C07286=1082.172,307.189,411.754,175.899,25.836,154.334
C07287=1082.167,306.941,411.785,175.896,25.832,154.333
C07288=1082.161,306.693,411.817,175.893,25.828,154.332
C07289=1082.155,306.445,411.848,175.890,25.824,154.332
C07290=1082.150,306.197,411.879,175.887,25.820,154.331
C07291=1082.144,305.949,411.911,175.885,25.816,154.331
C07292=1082.138,305.702,411.942,175.882,25.812,154.330
C07293=1082.132,305.453,411.973,175.879,25.808,154.330
C07294=1082.126,305.206,412.004,175.876,25.804,154.329
C07295=1082.121,304.958,412.036,175.873,25.800,154.328
C07296=1082.115,304.709,412.067,175.870,25.796,154.328
C07297=1082.109,304.462,412.098,175.867,25.792,154.327
C07298=1082.103,304.213,412.130,175.863,25.788,154.327
C07299=1082.093,303.800,412.182,175.859,25.781,154.326
C07300=1082.084,303.388,412.233,175.855,25.775,154.325
C07301=1082.075,302.974,412.286,175.849,25.768,154.324
C07302=1082.065,302.561,412.338,175.845,25.762,154.323
C07303=1082.059,302.314,412.368,175.842,25.758,154.323
C07304=1082.053,302.065,412.400,175.839,25.753,154.322
C07305=1082.047,301.818,412.430,175.836,25.749,154.321
C07306=1082.042,301.570,412.462,175.833,25.746,154.321
C07307=1082.037,301.322,412.493,175.831,25.742,154.320
C07308=1082.031,301.073,412.524,175.828,25.738,154.320
C07309=1082.025,300.826,412.555,175.825,25.734,154.319
C07310=1082.019,300.578,412.586,175.822,25.730,154.319
C07311=1082.014,300.330,412.617,175.818,25.726,154.318
C07312=1082.008,300.082,412.648,175.815,25.722,154.318
C07313=1082.002,299.834,412.679,175.813,25.718,154.317
C07314=1081.997,299.586,412.709,175.810,25.714,154.317
C07315=1081.991,299.339,412.741,175.807,25.710,154.316
C07316=1081.985,299.090,412.772,175.804,25.706,154.315
C07317=1081.980,298.842,412.803,175.801,25.702,154.315
C07318=1081.974,298.594,412.833,175.798,25.698,154.314
C07319=1081.969,298.346,412.864,175.796,25.695,154.314
C07320=1081.963,298.099,412.895,175.793,25.690,154.313
C07321=1081.957,297.850,412.926,175.790,25.686,154.313
C07322=1081.951,297.602,412.957,175.787,25.682,154.312
C07323=1081.945,297.354,412.987,175.784,25.678,154.312
C07324=1081.940,297.106,413.017,175.782,25.675,154.311
C07325=1081.934,296.858,413.049,175.779,25.671,154.310
C07326=1081.928,296.610,413.079,175.776,25.667,154.310
C07327=1081.922,296.362,413.109,175.773,25.663,154.309
C07328=1081.916,296.114,413.140,175.771,25.660,154.309
C07329=1081.910,295.866,413.172,175.767,25.656,154.308
C07330=1081.905,295.618,413.202,175.764,25.652,154.308
C07331=1081.899,295.370,413.232,175.761,25.648,154.307
C07332=1081.893,295.122,413.263,175.758,25.644,154.307
C07333=1081.887,294.875,413.293,175.756,25.641,154.306
C07334=1081.881,294.625,413.323,175.753,25.637,154.306
C07335=1081.875,294.378,413.353,175.750,25.633,154.305
C07336=1081.870,294.130,413.384,175.747,25.629,154.305
C07337=1081.864,293.882,413.415,175.744,25.625,154.304
C07338=1081.859,293.634,413.445,175.742,25.621,154.304
C07339=1081.853,293.386,413.475,175.739,25.618,154.303
C07340=1081.846,293.138,413.506,175.736,25.614,154.303
C07341=1081.841,292.890,413.537,175.733,25.610,154.302
C07342=1081.835,292.642,413.567,175.730,25.607,154.302
C07343=1081.829,292.393,413.597,175.727,25.603,154.301
C07344=1081.824,292.145,413.627,175.724,25.599,154.301
C07345=1081.818,291.897,413.658,175.721,25.595,154.300
C07346=1081.812,291.650,413.688,175.719,25.591,154.300
C07347=1081.806,291.401,413.719,175.716,25.588,154.299
C07348=1081.801,291.153,413.749,175.713,25.584,154.299
C07349=1081.795,290.905,413.779,175.710,25.580,154.298
C07350=1081.789,290.657,413.809,175.708,25.576,154.298
C07351=1081.780,290.258,413.858,175.703,25.570,154.297
C07352=1081.771,289.859,413.906,175.699,25.564,154.296
C07353=1081.761,289.460,413.955,175.694,25.558,154.295
C07354=1081.751,289.062,414.003,175.690,25.552,154.294
C07355=1081.746,288.813,414.032,175.687,25.548,154.294
C07356=1081.740,288.565,414.063,175.684,25.545,154.294
C07357=1081.734,288.318,414.093,175.681,25.541,154.293
C07358=1081.729,288.069,414.123,175.679,25.537,154.292
C07359=1081.723,287.821,414.153,175.675,25.533,154.292
C07360=1081.717,287.573,414.182,175.672,25.530,154.292
C07361=1081.711,287.325,414.212,175.670,25.526,154.291
C07362=1081.705,287.077,414.242,175.667,25.522,154.290
C07363=1081.699,286.829,414.272,175.664,25.519,154.290
C07364=1081.694,286.581,414.302,175.661,25.515,154.290
C07365=1081.688,286.333,414.332,175.659,25.511,154.289
C07366=1081.682,286.085,414.362,175.656,25.507,154.288
C07367=1081.676,285.837,414.392,175.653,25.504,154.288
C07368=1081.670,285.589,414.421,175.651,25.500,154.288
C07369=1081.665,285.340,414.451,175.648,25.496,154.287
C07370=1081.659,285.092,414.481,175.644,25.493,154.287
C07371=1081.653,284.844,414.511,175.641,25.489,154.286
C07372=1081.647,284.596,414.540,175.639,25.485,154.286
C07373=1081.642,284.348,414.571,175.636,25.482,154.285
C07374=1081.636,284.099,414.600,175.633,25.478,154.285
C07375=1081.631,283.851,414.630,175.631,25.474,154.284
C07376=1081.624,283.603,414.660,175.628,25.471,154.284
C07377=1081.618,283.355,414.689,175.625,25.467,154.283
C07378=1081.613,283.107,414.719,175.623,25.463,154.283
C07379=1081.607,282.859,414.749,175.620,25.460,154.282
C07380=1081.601,282.611,414.778,175.617,25.456,154.282
C07381=1081.595,282.362,414.808,175.614,25.452,154.281
C07382=1081.590,282.114,414.837,175.611,25.449,154.281
C07383=1081.584,281.865,414.867,175.608,25.445,154.280
C07384=1081.578,281.619,414.896,175.606,25.441,154.280
C07385=1081.573,281.370,414.926,175.603,25.438,154.279
C07386=1081.567,281.122,414.956,175.600,25.434,154.279
C07387=1081.561,280.873,414.985,175.598,25.430,154.278
C07388=1081.556,280.625,415.014,175.595,25.427,154.278
C07389=1081.550,280.377,415.044,175.592,25.423,154.277
C07390=1081.544,280.128,415.073,175.590,25.419,154.277
C07391=1081.538,279.881,415.103,175.587,25.416,154.276
C07392=1081.532,279.633,415.132,175.584,25.412,154.276
C07393=1081.526,279.384,415.162,175.581,25.408,154.275
C07394=1081.521,279.137,415.191,175.578,25.405,154.275
C07395=1081.515,278.888,415.220,175.575,25.401,154.274
C07396=1081.509,278.640,415.249,175.573,25.398,154.274
C07397=1081.503,278.392,415.279,175.570,25.394,154.274
C07398=1081.498,278.143,415.309,175.567,25.390,154.273
C07399=1081.492,277.895,415.338,175.565,25.387,154.273
C07400=1081.486,277.647,415.367,175.562,25.383,154.272
C07401=1081.481,277.399,415.395,175.559,25.379,154.272
C07402=1081.475,277.150,415.425,175.557,25.376,154.271
C07403=1081.466,276.762,415.471,175.552,25.370,154.270
C07404=1081.457,276.373,415.516,175.547,25.364,154.270
C07405=1081.448,275.983,415.562,175.544,25.359,154.269
C07406=1081.438,275.594,415.608,175.539,25.353,154.268
C07407=1081.434,275.346,415.637,175.536,25.349,154.268
C07408=1081.427,275.097,415.666,175.534,25.346,154.267
C07409=1081.421,274.849,415.695,175.531,25.342,154.267
C07410=1081.416,274.601,415.725,175.528,25.339,154.266
C07411=1081.410,274.353,415.753,175.526,25.335,154.266
C07412=1081.405,274.104,415.782,175.523,25.331,154.265
C07413=1081.399,273.856,415.811,175.520,25.328,154.265
C07414=1081.392,273.608,415.840,175.517,25.324,154.264
C07415=1081.388,273.360,415.869,175.514,25.321,154.264
C07416=1081.381,273.112,415.898,175.512,25.317,154.264
C07417=1081.375,272.863,415.927,175.509,25.314,154.263
C07418=1081.370,272.614,415.956,175.507,25.311,154.263
C07419=1081.364,272.367,415.984,175.504,25.307,154.262
C07420=1081.358,272.119,416.013,175.501,25.303,154.262
C07421=1081.352,271.870,416.042,175.499,25.300,154.261
C07422=1081.347,271.622,416.071,175.496,25.296,154.261
C07423=1081.341,271.374,416.100,175.493,25.292,154.260
C07424=1081.335,271.125,416.128,175.490,25.289,154.260
C07425=1081.329,270.877,416.157,175.487,25.285,154.259
C07426=1081.324,270.629,416.186,175.485,25.282,154.259
C07427=1081.318,270.381,416.215,175.482,25.278,154.259
C07428=1081.312,270.132,416.243,175.480,25.275,154.258
C07429=1081.306,269.885,416.272,175.477,25.271,154.258
C07430=1081.301,269.636,416.301,175.474,25.267,154.257
C07431=1081.295,269.387,416.330,175.472,25.264,154.257
C07432=1081.290,269.139,416.358,175.469,25.260,154.256
C07433=1081.283,268.891,416.387,175.466,25.257,154.256
C07434=1081.277,268.643,416.415,175.463,25.253,154.255
C07435=1081.272,268.394,416.443,175.460,25.250,154.255
C07436=1081.266,268.146,416.472,175.458,25.247,154.255
C07437=1081.261,267.897,416.501,175.455,25.243,154.254
C07438=1081.255,267.650,416.530,175.453,25.240,154.254
C07439=1081.249,267.401,416.558,175.450,25.236,154.253
C07440=1081.243,267.152,416.587,175.448,25.232,154.253
C07441=1081.237,266.905,416.615,175.445,25.229,154.252
C07442=1081.231,266.656,416.644,175.442,25.225,154.252
C07443=1081.226,266.408,416.672,175.439,25.222,154.251
C07444=1081.220,266.160,416.701,175.436,25.218,154.251
C07445=1081.214,265.911,416.729,175.434,25.215,154.250
C07446=1081.209,265.663,416.757,175.431,25.211,154.250
C07447=1081.203,265.414,416.785,175.429,25.208,154.250
C07448=1081.198,265.167,416.814,175.426,25.204,154.249
C07449=1081.192,264.918,416.843,175.424,25.201,154.249
C07450=1081.186,264.670,416.871,175.421,25.197,154.248
C07451=1081.180,264.421,416.899,175.418,25.193,154.248
C07452=1081.175,264.173,416.927,175.415,25.190,154.247
C07453=1081.169,263.924,416.955,175.412,25.186,154.247
C07454=1081.162,263.677,416.984,175.410,25.183,154.246
C07455=1081.154,263.290,417.027,175.406,25.178,154.246
C07456=1081.145,262.904,417.071,175.402,25.172,154.245
C07457=1081.135,262.518,417.115,175.397,25.167,154.244
C07458=1081.126,262.132,417.159,175.394,25.162,154.244
C07459=1081.120,261.883,417.187,175.390,25.158,154.243
C07460=1081.115,261.635,417.215,175.388,25.155,154.243
C07461=1081.108,261.387,417.243,175.385,25.151,154.242
C07462=1081.103,261.139,417.271,175.383,25.148,154.242
C07463=1081.097,260.890,417.299,175.380,25.144,154.242
C07464=1081.092,260.642,417.327,175.378,25.141,154.241
C07465=1081.085,260.393,417.355,175.375,25.137,154.241
C07466=1081.079,260.145,417.383,175.372,25.134,154.240
C07467=1081.074,259.897,417.411,175.370,25.131,154.240
C07468=1081.068,259.649,417.439,175.366,25.127,154.240
C07469=1081.062,259.400,417.467,175.364,25.124,154.239
C07470=1081.056,259.152,417.494,175.361,25.120,154.239
C07471=1081.051,258.903,417.522,175.359,25.117,154.238
C07472=1081.045,258.655,417.550,175.356,25.113,154.238
C07473=1081.039,258.406,417.578,175.354,25.110,154.237
C07474=1081.033,258.158,417.606,175.351,25.106,154.237
C07475=1081.027,257.909,417.634,175.349,25.103,154.236
C07476=1081.021,257.662,417.661,175.346,25.099,154.236
C07477=1081.016,257.412,417.689,175.343,25.096,154.236
C07478=1081.010,257.164,417.717,175.340,25.093,154.235
C07479=1081.004,256.916,417.745,175.338,25.089,154.235
C07480=1080.998,256.668,417.773,175.335,25.085,154.234
C07481=1080.993,256.419,417.800,175.333,25.082,154.234
C07482=1080.986,256.171,417.828,175.330,25.079,154.233
C07483=1080.981,255.923,417.856,175.328,25.075,154.233
C07484=1080.975,255.674,417.884,175.325,25.072,154.233
C07485=1080.969,255.426,417.911,175.322,25.068,154.232
C07486=1080.964,255.178,417.939,175.319,25.065,154.232
C07487=1080.958,254.929,417.967,175.317,25.061,154.231
C07488=1080.952,254.680,417.994,175.314,25.058,154.231
C07489=1080.946,254.432,418.022,175.312,25.055,154.230
C07490=1080.941,254.183,418.049,175.309,25.051,154.230
C07491=1080.935,253.935,418.077,175.307,25.048,154.229
C07492=1080.929,253.686,418.105,175.304,25.044,154.229
C07493=1080.924,253.438,418.132,175.302,25.041,154.229
C07494=1080.918,253.190,418.159,175.299,25.037,154.228
C07495=1080.913,252.941,418.187,175.296,25.034,154.228
C07496=1080.906,252.693,418.214,175.294,25.031,154.227
C07497=1080.901,252.444,418.242,175.291,25.027,154.227
C07498=1080.896,252.196,418.270,175.289,25.023,154.226
C07499=1080.890,251.947,418.297,175.286,25.020,154.226
C07500=1080.884,251.699,418.325,175.284,25.016,154.226
C07501=1080.879,251.451,418.351,175.281,25.013,154.225
C07502=1080.873,251.202,418.380,175.279,25.010,154.225
C07503=1080.868,250.953,418.407,175.276,25.006,154.224
C07504=1080.862,250.706,418.434,175.273,25.003,154.224
C07505=1080.857,250.457,418.461,175.270,24.999,154.223
C07506=1080.850,250.208,418.489,175.268,24.995,154.223
C07507=1080.842,249.820,418.532,175.265,24.990,154.222
C07508=1080.833,249.431,418.574,175.260,24.985,154.222
C07509=1080.824,249.042,418.617,175.256,24.979,154.221
C07510=1080.815,248.654,418.660,175.252,24.974,154.220
C07511=1080.810,248.404,418.687,175.250,24.970,154.220
C07512=1080.804,248.156,418.714,175.247,24.966,154.219
C07513=1080.799,247.908,418.742,175.245,24.963,154.219
C07514=1080.793,247.659,418.769,175.242,24.960,154.218
C07515=1080.788,247.411,418.796,175.239,24.956,154.218
C07516=1080.782,247.162,418.823,175.237,24.953,154.217
C07517=1080.776,246.914,418.851,175.234,24.949,154.217
C07518=1080.770,246.665,418.878,175.232,24.946,154.217
C07519=1080.765,246.417,418.904,175.229,24.942,154.216
C07520=1080.759,246.168,418.931,175.227,24.939,154.216
C07521=1080.754,245.920,418.958,175.225,24.936,154.215
C07522=1080.747,245.671,418.985,175.222,24.932,154.215
C07523=1080.742,245.423,419.013,175.220,24.929,154.214
C07524=1080.736,245.174,419.040,175.217,24.925,154.214
C07525=1080.730,244.926,419.066,175.214,24.922,154.214
C07526=1080.725,244.677,419.094,175.211,24.918,154.213
C07527=1080.720,244.429,419.120,175.209,24.915,154.213
C07528=1080.713,244.180,419.147,175.207,24.912,154.212
C07529=1080.707,243.932,419.174,175.204,24.908,154.212
C07530=1080.702,243.683,419.201,175.202,24.905,154.211
C07531=1080.697,243.435,419.228,175.199,24.901,154.211
C07532=1080.691,243.186,419.254,175.197,24.898,154.211
C07533=1080.686,242.937,419.282,175.194,24.895,154.210
C07534=1080.680,242.689,419.308,175.192,24.891,154.210
C07535=1080.674,242.441,419.335,175.189,24.888,154.209
C07536=1080.668,242.192,419.362,175.186,24.884,154.209
C07537=1080.662,241.943,419.389,175.184,24.881,154.209
C07538=1080.656,241.695,419.415,175.182,24.878,154.208
C07539=1080.651,241.447,419.442,175.179,24.874,154.208
C07540=1080.645,241.198,419.469,175.177,24.871,154.207
C07541=1080.640,240.950,419.496,175.174,24.867,154.207
C07542=1080.634,240.701,419.522,175.172,24.864,154.206
C07543=1080.628,240.453,419.549,175.169,24.861,154.206
C07544=1080.622,240.204,419.576,175.166,24.857,154.206
C07545=1080.616,239.955,419.602,175.164,24.853,154.205
C07546=1080.611,239.706,419.629,175.161,24.850,154.205
C07547=1080.605,239.458,419.655,175.159,24.847,154.204
C07548=1080.599,239.210,419.682,175.157,24.844,154.204
C07549=1080.593,238.961,419.709,175.154,24.840,154.204
C07550=1080.588,238.712,419.735,175.152,24.836,154.203
C07551=1080.582,238.464,419.761,175.150,24.833,154.203
C07552=1080.576,238.216,419.788,175.146,24.830,154.202
C07553=1080.571,237.967,419.815,175.144,24.827,154.202
C07554=1080.565,237.719,419.841,175.141,24.823,154.201
C07555=1080.559,237.470,419.867,175.139,24.820,154.201
C07556=1080.554,237.222,419.894,175.137,24.816,154.200
C07557=1080.548,236.973,419.920,175.134,24.813,154.200
C07558=1080.542,236.724,419.946,175.132,24.810,154.200
C07559=1080.533,236.329,419.989,175.128,24.804,154.199
C07560=1080.524,235.934,420.031,175.124,24.799,154.198
C07561=1080.515,235.538,420.073,175.120,24.793,154.198
C07562=1080.506,235.142,420.115,175.116,24.788,154.197
C07563=1080.500,234.893,420.141,175.113,24.784,154.197
C07564=1080.495,234.645,420.168,175.111,24.781,154.196
C07565=1080.489,234.396,420.194,175.108,24.777,154.196
C07566=1080.483,234.147,420.220,175.106,24.774,154.195
C07567=1080.478,233.899,420.246,175.104,24.771,154.195
C07568=1080.472,233.651,420.272,175.101,24.767,154.194
C07569=1080.466,233.402,420.298,175.099,24.764,154.194
C07570=1080.461,233.154,420.324,175.097,24.760,154.194
C07571=1080.455,232.905,420.350,175.094,24.757,154.193
C07572=1080.449,232.656,420.377,175.092,24.754,154.193
C07573=1080.444,232.407,420.403,175.089,24.751,154.192
C07574=1080.438,232.159,420.430,175.086,24.747,154.192
C07575=1080.432,231.910,420.455,175.084,24.743,154.191
C07576=1080.426,231.662,420.482,175.082,24.740,154.191
C07577=1080.421,231.413,420.508,175.079,24.737,154.191
C07578=1080.415,231.164,420.533,175.077,24.734,154.190
C07579=1080.410,230.916,420.560,175.075,24.730,154.190
C07580=1080.404,230.668,420.585,175.072,24.726,154.189
C07581=1080.398,230.419,420.612,175.070,24.723,154.189
C07582=1080.393,230.170,420.638,175.067,24.720,154.188
C07583=1080.387,229.921,420.664,175.064,24.716,154.188
C07584=1080.381,229.673,420.690,175.062,24.713,154.188
C07585=1080.375,229.424,420.716,175.060,24.710,154.187
C07586=1080.369,229.176,420.741,175.057,24.706,154.187
C07587=1080.364,228.927,420.767,175.055,24.703,154.186
C07588=1080.358,228.678,420.793,175.053,24.700,154.186
C07589=1080.352,228.430,420.818,175.051,24.696,154.186
C07590=1080.347,228.181,420.844,175.048,24.693,154.185
C07591=1080.341,227.932,420.870,175.045,24.690,154.185
C07592=1080.335,227.684,420.896,175.043,24.687,154.184
C07593=1080.329,227.435,420.922,175.040,24.683,154.184
C07594=1080.323,227.187,420.948,175.038,24.679,154.183
C07595=1080.318,226.938,420.973,175.036,24.676,154.183
C07596=1080.313,226.689,420.999,175.033,24.673,154.183
C07597=1080.307,226.441,421.024,175.031,24.669,154.182
C07598=1080.301,226.192,421.051,175.029,24.666,154.182
C07599=1080.295,225.944,421.076,175.027,24.663,154.181
C07600=1080.289,225.695,421.102,175.024,24.659,154.181
C07601=1080.283,225.447,421.127,175.022,24.656,154.181
C07602=1080.278,225.198,421.153,175.019,24.653,154.180
C07603=1080.273,224.949,421.179,175.016,24.649,154.180
C07604=1080.266,224.700,421.205,175.014,24.645,154.179
C07605=1080.261,224.452,421.230,175.012,24.642,154.179
C07606=1080.255,224.203,421.255,175.010,24.639,154.178
C07607=1080.250,223.954,421.281,175.007,24.636,154.178
C07608=1080.244,223.705,421.307,175.005,24.632,154.178
C07609=1080.239,223.457,421.332,175.003,24.629,154.177
C07610=1080.232,223.208,421.358,175.000,24.625,154.177
C07611=1080.224,222.805,421.399,174.996,24.620,154.176
C07612=1080.214,222.400,421.441,174.993,24.614,154.175
C07613=1080.205,221.996,421.483,174.988,24.609,154.175
C07614=1080.196,221.592,421.524,174.985,24.603,154.174
C07615=1080.190,221.343,421.550,174.982,24.600,154.174
C07616=1080.184,221.095,421.575,174.980,24.597,154.173
C07617=1080.179,220.847,421.600,174.977,24.593,154.173
C07618=1080.173,220.597,421.625,174.975,24.590,154.172
C07619=1080.167,220.349,421.651,174.973,24.587,154.172
C07620=1080.161,220.100,421.676,174.971,24.583,154.172
C07621=1080.155,219.852,421.701,174.968,24.580,154.171
C07622=1080.150,219.603,421.727,174.966,24.577,154.171
C07623=1080.144,219.354,421.752,174.964,24.573,154.170
C07624=1080.139,219.106,421.776,174.962,24.570,154.170
C07625=1080.133,218.857,421.802,174.959,24.566,154.169
C07626=1080.127,218.608,421.828,174.956,24.563,154.169
C07627=1080.121,218.360,421.853,174.954,24.560,154.169
C07628=1080.116,218.110,421.878,174.952,24.557,154.168
C07629=1080.110,217.862,421.903,174.949,24.553,154.168
C07630=1080.104,217.614,421.928,174.947,24.549,154.167
C07631=1080.098,217.365,421.953,174.945,24.546,154.167
C07632=1080.093,217.116,421.979,174.943,24.543,154.166
C07633=1080.087,216.868,422.004,174.940,24.539,154.166
C07634=1080.081,216.618,422.028,174.938,24.536,154.166
C07635=1080.076,216.370,422.053,174.936,24.533,154.165
C07636=1080.070,216.121,422.079,174.934,24.529,154.165
C07637=1080.064,215.872,422.104,174.930,24.526,154.164
C07638=1080.059,215.624,422.129,174.928,24.523,154.164
C07639=1080.053,215.375,422.154,174.926,24.519,154.164
C07640=1080.048,215.127,422.179,174.924,24.516,154.163
C07641=1080.042,214.878,422.204,174.921,24.512,154.163
C07642=1080.037,214.629,422.229,174.919,24.509,154.162
C07643=1080.030,214.381,422.254,174.917,24.506,154.162
C07644=1080.024,214.131,422.279,174.915,24.503,154.161
C07645=1080.020,213.883,422.304,174.913,24.499,154.161
C07646=1080.013,213.634,422.329,174.910,24.495,154.161
C07647=1080.008,213.386,422.354,174.908,24.492,154.160
C07648=1080.002,213.137,422.379,174.905,24.489,154.160
C07649=1079.997,212.889,422.403,174.903,24.486,154.159
C07650=1079.991,212.639,422.428,174.900,24.482,154.159
C07651=1079.986,212.391,422.453,174.898,24.478,154.158
C07652=1079.980,212.142,422.478,174.896,24.475,154.158
C07653=1079.974,211.894,422.503,174.894,24.472,154.158
C07654=1079.968,211.644,422.528,174.892,24.469,154.157
C07655=1079.963,211.396,422.553,174.889,24.465,154.157
C07656=1079.957,211.147,422.577,174.887,24.461,154.156
C07657=1079.952,210.899,422.602,174.885,24.458,154.156
C07658=1079.945,210.650,422.627,174.883,24.455,154.156
C07659=1079.940,210.401,422.651,174.881,24.452,154.155
C07660=1079.934,210.152,422.676,174.877,24.448,154.155
C07661=1079.929,209.904,422.701,174.875,24.445,154.154
C07662=1079.923,209.655,422.725,174.873,24.441,154.154
C07663=1079.913,209.254,422.765,174.870,24.436,154.153
C07664=1079.905,208.855,422.804,174.866,24.431,154.153
C07665=1079.895,208.455,422.844,174.863,24.425,154.152
C07666=1079.886,208.055,422.884,174.859,24.420,154.151
C07667=1079.863,207.021,422.983,174.758,24.366,154.153
C07668=1079.856,206.772,423.007,174.755,24.364,154.153
C07669=1079.851,206.523,423.031,174.753,24.361,154.152
C07670=1079.846,206.275,423.056,174.750,24.359,154.152
C07671=1079.841,206.026,423.080,174.748,24.357,154.152
C07672=1079.834,205.776,423.103,174.746,24.354,154.152
C07673=1079.829,205.528,423.128,174.743,24.352,154.152
C07674=1079.824,205.279,423.152,174.740,24.349,154.151
C07675=1079.818,205.031,423.175,174.738,24.347,154.151
C07676=1079.813,204.782,423.199,174.735,24.344,154.151
C07677=1079.807,204.532,423.224,174.733,24.342,154.151
C07678=1079.801,204.284,423.247,174.731,24.339,154.151
C07679=1079.796,204.035,423.271,174.728,24.337,154.150
C07680=1079.790,203.787,423.294,174.726,24.334,154.150
C07681=1079.784,203.538,423.319,174.724,24.332,154.150
C07682=1079.779,203.289,423.342,174.721,24.329,154.150
C07683=1079.773,203.040,423.366,174.719,24.327,154.150
C07684=1079.767,202.791,423.391,174.717,24.325,154.149
C07685=1079.762,202.542,423.414,174.714,24.322,154.149
C07686=1079.756,202.294,423.438,174.712,24.320,154.149
C07687=1079.750,202.046,423.461,174.710,24.318,154.149
C07688=1079.745,201.796,423.485,174.707,24.315,154.149
C07689=1079.739,201.547,423.509,174.705,24.313,154.148
C07690=1079.734,201.298,423.533,174.702,24.310,154.148
C07691=1079.728,201.050,423.556,174.700,24.308,154.148
C07692=1079.722,200.801,423.579,174.698,24.306,154.148
C07693=1079.717,200.552,423.603,174.695,24.303,154.148
C07694=1079.710,200.303,423.627,174.693,24.301,154.147
C07695=1079.705,200.054,423.651,174.690,24.299,154.147
C07696=1079.699,199.805,423.674,174.688,24.296,154.147
C07697=1079.693,199.557,423.698,174.686,24.294,154.147
C07698=1079.688,199.308,423.721,174.683,24.292,154.147
C07699=1079.682,199.060,423.745,174.681,24.289,154.146
C07700=1079.677,198.810,423.768,174.679,24.287,154.146
C07701=1079.671,198.561,423.792,174.676,24.285,154.146
C07702=1079.665,198.313,423.815,174.674,24.282,154.146
C07703=1079.660,198.063,423.839,174.672,24.280,154.146
C07704=1079.654,197.815,423.862,174.669,24.278,154.146
C07705=1079.648,197.566,423.885,174.667,24.275,154.145
C07706=1079.643,197.318,423.910,174.664,24.273,154.145
C07707=1079.637,197.069,423.933,174.662,24.271,154.145
C07708=1079.631,196.820,423.956,174.660,24.268,154.145
C07709=1079.626,196.571,423.980,174.657,24.266,154.145
C07710=1079.620,196.322,424.003,174.655,24.264,154.145
C07711=1079.615,196.073,424.026,174.653,24.261,154.144
C07712=1079.609,195.824,424.050,174.650,24.259,154.144
C07713=1079.603,195.575,424.073,174.648,24.256,154.144
C07714=1079.597,195.326,424.096,174.646,24.255,154.144
C07715=1079.592,195.078,424.121,174.644,24.252,154.144
C07716=1079.586,194.829,424.143,174.642,24.250,154.143
C07717=1079.580,194.580,424.166,174.639,24.247,154.143
C07718=1079.575,194.331,424.189,174.637,24.245,154.143
C07719=1079.569,194.082,424.214,174.635,24.243,154.143
C07720=1079.564,193.834,424.237,174.632,24.240,154.143
C07721=1079.558,193.585,424.259,174.630,24.238,154.142
C07722=1079.553,193.335,424.283,174.628,24.236,154.142
C07723=1079.547,193.087,424.306,174.625,24.233,154.142
C07724=1079.541,192.838,424.330,174.623,24.231,154.142
C07725=1079.535,192.589,424.353,174.620,24.229,154.142
C07726=1079.530,192.340,424.376,174.618,24.226,154.141
C07727=1079.525,192.091,424.399,174.616,24.224,154.141
C07728=1079.519,191.812,424.425,174.614,24.221,154.141
C07729=1079.512,191.532,424.451,174.611,24.218,154.141
C07730=1079.506,191.252,424.477,174.608,24.216,154.141
C07731=1079.500,190.972,424.503,174.606,24.213,154.140
C07732=1079.494,190.723,424.526,174.603,24.211,154.140
C07733=1079.489,190.475,424.549,174.601,24.208,154.140
C07734=1079.484,190.226,424.573,174.599,24.206,154.140
C07735=1079.478,189.977,424.595,174.596,24.203,154.139
C07736=1079.472,189.728,424.618,174.595,24.201,154.139
C07737=1079.467,189.479,424.641,174.593,24.199,154.139
C07738=1079.462,189.230,424.665,174.590,24.197,154.139
C07739=1079.456,188.981,424.688,174.588,24.194,154.139
C07740=1079.450,188.732,424.711,174.585,24.192,154.138
C07741=1079.444,188.483,424.734,174.583,24.189,154.138
C07742=1079.439,188.235,424.756,174.581,24.187,154.138
C07743=1079.434,187.986,424.780,174.578,24.185,154.138
C07744=1079.429,187.737,424.803,174.576,24.182,154.138
C07745=1079.423,187.488,424.826,174.574,24.180,154.137
C07746=1079.417,187.239,424.849,174.572,24.177,154.137
C07747=1079.411,186.990,424.872,174.570,24.175,154.137
C07748=1079.406,186.741,424.895,174.568,24.172,154.137
C07749=1079.401,186.493,424.918,174.565,24.170,154.137
C07750=1079.396,186.244,424.941,174.563,24.168,154.136
C07751=1079.390,185.995,424.964,174.561,24.165,154.136
C07752=1079.384,185.746,424.987,174.558,24.163,154.136
C07753=1079.379,185.496,425.009,174.556,24.161,154.136
C07754=1079.374,185.248,425.031,174.554,24.159,154.136
C07755=1079.369,184.999,425.055,174.552,24.156,154.135
C07756=1079.362,184.750,425.077,174.550,24.154,154.135
C07757=1079.356,184.502,425.100,174.547,24.152,154.135
C07758=1079.351,184.253,425.123,174.545,24.149,154.135
C07759=1079.345,184.003,425.145,174.543,24.147,154.135
C07760=1079.339,183.754,425.168,174.540,24.145,154.135
C07761=1079.333,183.506,425.191,174.538,24.142,154.134
C07762=1079.327,183.257,425.214,174.536,24.140,154.134
C07763=1079.322,183.007,425.236,174.534,24.138,154.134
C07764=1079.317,182.759,425.258,174.532,24.136,154.134
C07765=1079.310,182.510,425.281,174.529,24.133,154.134
C07766=1079.305,182.262,425.304,174.527,24.131,154.133
C07767=1079.299,182.012,425.326,174.525,24.129,154.133
C07768=1079.293,181.763,425.349,174.523,24.127,154.133
C07769=1079.288,181.514,425.372,174.521,24.125,154.133
C07770=1079.281,181.265,425.394,174.518,24.122,154.133
C07771=1079.276,181.016,425.416,174.516,24.120,154.133
C07772=1079.271,180.768,425.439,174.514,24.118,154.132
C07773=1079.264,180.519,425.461,174.511,24.115,154.132
C07774=1079.259,180.270,425.484,174.509,24.113,154.132
C07775=1079.253,180.021,425.507,174.507,24.111,154.132
C07776=1079.248,179.771,425.529,174.505,24.109,154.132
C07777=1079.241,179.523,425.551,174.503,24.106,154.131
C07778=1079.236,179.274,425.573,174.500,24.104,154.131
C07779=1079.231,179.025,425.596,174.498,24.102,154.131
C07780=1079.225,178.776,425.619,174.497,24.099,154.131
C07781=1079.219,178.527,425.641,174.494,24.097,154.131
C07782=1079.214,178.279,425.663,174.492,24.095,154.131
C07783=1079.208,178.029,425.685,174.489,24.093,154.130
C07784=1079.202,177.781,425.708,174.487,24.090,154.130
C07785=1079.196,177.531,425.730,174.485,24.088,154.130
C07786=1079.190,177.282,425.753,174.483,24.086,154.130
C07787=1079.185,177.034,425.774,174.481,24.083,154.130
C07788=1079.179,176.785,425.797,174.479,24.081,154.129
C07789=1079.174,176.535,425.819,174.476,24.079,154.129
C07790=1079.167,176.287,425.842,174.474,24.076,154.129
C07791=1079.162,176.038,425.864,174.472,24.074,154.129
C07792=1079.156,175.757,425.889,174.469,24.071,154.129
C07793=1079.149,175.478,425.913,174.467,24.069,154.129
C07794=1079.143,175.197,425.939,174.465,24.066,154.128
C07795=1079.137,174.917,425.964,174.462,24.064,154.128
C07796=1079.131,174.668,425.986,174.460,24.061,154.128
C07797=1079.126,174.419,426.008,174.458,24.059,154.128
C07798=1079.120,174.170,426.030,174.456,24.057,154.127
C07799=1079.114,173.921,426.053,174.454,24.055,154.127
C07800=1079.109,173.672,426.075,174.452,24.052,154.127
C07801=1079.103,173.424,426.097,174.449,24.050,154.127
C07802=1079.097,173.174,426.119,174.447,24.048,154.127
C07803=1079.092,172.926,426.141,174.445,24.045,154.126
C07804=1079.086,172.677,426.163,174.443,24.043,154.126
C07805=1079.081,172.427,426.186,174.441,24.041,154.126
C07806=1079.076,172.179,426.207,174.438,24.038,154.126
C07807=1079.070,171.929,426.229,174.437,24.036,154.126
C07808=1079.064,171.680,426.252,174.435,24.034,154.125
C07809=1079.059,171.432,426.274,174.432,24.031,154.125
C07810=1079.053,171.182,426.296,174.430,24.029,154.125
C07811=1079.048,170.934,426.317,174.428,24.027,154.125
C07812=1079.042,170.685,426.340,174.426,24.025,154.125
C07813=1079.036,170.436,426.362,174.424,24.022,154.124
C07814=1079.031,170.187,426.383,174.421,24.020,154.124
C07815=1079.025,169.938,426.405,174.419,24.017,154.124
C07816=1079.020,169.689,426.428,174.418,24.015,154.124
C07817=1079.014,169.440,426.450,174.415,24.013,154.124
C07818=1079.008,169.191,426.472,174.413,24.010,154.123
C07819=1079.003,168.942,426.493,174.411,24.008,154.123
C07820=1078.997,168.693,426.515,174.409,24.006,154.123
C07821=1078.992,168.444,426.537,174.407,24.004,154.123
C07822=1078.986,168.195,426.560,174.405,24.001,154.123
C07823=1078.981,167.946,426.581,174.403,23.999,154.122
C07824=1078.975,167.697,426.603,174.401,23.996,154.122
C07825=1078.970,167.448,426.625,174.398,23.994,154.122
C07826=1078.964,167.199,426.647,174.396,23.991,154.122
C07827=1078.959,166.950,426.668,174.395,23.990,154.122
C07828=1078.953,166.701,426.690,174.392,23.987,154.121
C07829=1078.948,166.452,426.712,174.390,23.985,154.121
C07830=1078.942,166.203,426.734,174.388,23.982,154.121
C07831=1078.937,165.954,426.755,174.386,23.980,154.121
C07832=1078.931,165.705,426.777,174.384,23.977,154.121
C07833=1078.926,165.456,426.799,174.382,23.975,154.120
C07834=1078.920,165.207,426.821,174.379,23.973,154.120
C07835=1078.915,164.958,426.842,174.378,23.971,154.120
C07836=1078.909,164.709,426.864,174.376,23.968,154.120
C07837=1078.904,164.460,426.886,174.373,23.966,154.120
C07838=1078.898,164.211,426.908,174.372,23.963,154.119
C07839=1078.893,163.962,426.929,174.370,23.961,154.119
C07840=1078.887,163.713,426.951,174.367,23.958,154.119
C07841=1078.882,163.464,426.973,174.365,23.956,154.119
C07842=1078.876,163.215,426.995,174.364,23.954,154.118
C07843=1078.871,162.966,427.016,174.361,23.952,154.118
C07844=1078.866,162.718,427.038,174.359,23.949,154.118
C07845=1078.860,162.468,427.060,174.357,23.947,154.118
C07846=1078.855,162.220,427.081,174.355,23.944,154.118
C07847=1078.849,161.970,427.103,174.353,23.942,154.117
C07848=1078.844,161.721,427.124,174.351,23.940,154.117
C07849=1078.839,161.472,427.146,174.349,23.937,154.117
C07850=1078.833,161.223,427.168,174.347,23.935,154.117
C07851=1078.828,160.974,427.189,174.344,23.933,154.117
C07852=1078.821,160.725,427.210,174.343,23.930,154.116
C07853=1078.816,160.477,427.232,174.341,23.928,154.116
C07854=1078.811,160.227,427.253,174.338,23.926,154.116
C07855=1078.802,159.890,427.282,174.336,23.923,154.116
C07856=1078.797,159.632,427.304,174.334,23.921,154.115
C07857=1078.792,159.373,427.327,174.332,23.918,154.115
C07858=1078.785,159.114,427.348,174.329,23.916,154.115
C07859=1078.779,158.856,427.371,174.328,23.913,154.115
C07860=1078.774,158.607,427.393,174.325,23.911,154.115
C07861=1078.768,158.357,427.414,174.323,23.908,154.114
C07862=1078.762,158.109,427.435,174.322,23.907,154.114
C07863=1078.757,157.860,427.456,174.319,23.904,154.114
C07864=1078.751,157.610,427.477,174.317,23.902,154.114
C07865=1078.746,157.362,427.499,174.316,23.900,154.114
C07866=1078.740,157.112,427.521,174.313,23.897,154.113
C07867=1078.735,156.863,427.541,174.311,23.895,154.113
C07868=1078.729,156.615,427.562,174.310,23.893,154.113
C07869=1078.723,156.366,427.584,174.307,23.890,154.113
C07870=1078.718,156.116,427.605,174.305,23.888,154.113
C07871=1078.712,155.867,427.626,174.303,23.886,154.112
C07872=1078.706,155.619,427.648,174.301,23.883,154.112
C07873=1078.702,155.369,427.669,174.299,23.881,154.112
C07874=1078.695,155.120,427.690,174.297,23.879,154.112
C07875=1078.690,154.871,427.711,174.295,23.876,154.112
C07876=1078.684,154.622,427.733,174.293,23.874,154.111
C07877=1078.678,154.373,427.754,174.291,23.872,154.111
C07878=1078.673,154.124,427.774,174.289,23.869,154.111
C07879=1078.667,153.875,427.796,174.287,23.867,154.111
C07880=1078.662,153.626,427.817,174.285,23.865,154.111
C07881=1078.656,153.377,427.838,174.283,23.863,154.110
C07882=1078.650,153.128,427.859,174.281,23.860,154.110
C07883=1078.645,152.879,427.880,174.279,23.858,154.110
C07884=1078.639,152.630,427.901,174.277,23.855,154.110
C07885=1078.633,152.381,427.922,174.275,23.853,154.110
C07886=1078.628,152.132,427.943,174.273,23.851,154.109
C07887=1078.622,151.883,427.964,174.271,23.849,154.109
C07888=1078.617,151.633,427.985,174.270,23.846,154.109
C07889=1078.611,151.385,428.006,174.267,23.844,154.109
C07890=1078.606,151.136,428.027,174.265,23.841,154.108
C07891=1078.600,150.886,428.048,174.263,23.840,154.108
C07892=1078.594,150.637,428.069,174.261,23.837,154.108
C07893=1078.588,150.389,428.090,174.259,23.835,154.108
C07894=1078.582,150.139,428.111,174.257,23.832,154.108
C07895=1078.577,149.890,428.131,174.255,23.830,154.107
C07896=1078.571,149.642,428.152,174.254,23.828,154.107
C07897=1078.566,149.393,428.173,174.251,23.825,154.107
C07898=1078.560,149.143,428.194,174.249,23.823,154.107
C07899=1078.555,148.894,428.215,174.248,23.821,154.107
C07900=1078.549,148.645,428.236,174.245,23.818,154.106
C07901=1078.543,148.396,428.257,174.243,23.816,154.106
C07902=1078.538,148.147,428.278,174.242,23.814,154.106
C07903=1078.532,147.898,428.298,174.239,23.811,154.106
C07904=1078.527,147.649,428.318,174.238,23.810,154.106
C07905=1078.521,147.400,428.340,174.236,23.807,154.105
C07906=1078.515,147.150,428.361,174.233,23.805,154.105
C07907=1078.509,146.902,428.380,174.232,23.802,154.105
C07908=1078.503,146.652,428.402,174.229,23.800,154.105
C07909=1078.498,146.403,428.423,174.228,23.798,154.104
C07910=1078.493,146.154,428.443,174.226,23.795,154.104
C07911=1078.487,145.905,428.464,174.224,23.793,154.104
C07912=1078.481,145.656,428.485,174.222,23.791,154.104
C07913=1078.475,145.407,428.505,174.220,23.788,154.104
C07914=1078.470,145.158,428.526,174.218,23.786,154.103
C07915=1078.465,144.909,428.546,174.216,23.784,154.103
C07916=1078.458,144.659,428.567,174.214,23.781,154.103
C07917=1078.453,144.411,428.588,174.212,23.779,154.103
C07918=1078.447,144.162,428.609,174.210,23.777,154.103
C07919=1078.441,143.913,428.629,174.209,23.774,154.102
C07920=1078.435,143.632,428.652,174.206,23.772,154.102
C07921=1078.429,143.351,428.676,174.204,23.769,154.102
C07922=1078.423,143.070,428.699,174.202,23.767,154.102
C07923=1078.417,142.789,428.722,174.200,23.764,154.101
C07924=1078.411,142.540,428.742,174.197,23.761,154.101
C07925=1078.405,142.292,428.763,174.196,23.759,154.101
C07926=1078.400,142.042,428.784,174.194,23.757,154.101
C07927=1078.393,141.793,428.804,174.192,23.755,154.101
C07928=1078.388,141.544,428.824,174.190,23.752,154.100
C07929=1078.383,141.295,428.845,174.188,23.750,154.100
C07930=1078.377,141.046,428.865,174.186,23.748,154.100
C07931=1078.371,140.797,428.885,174.184,23.745,154.100
C07932=1078.366,140.548,428.906,174.183,23.743,154.099
C07933=1078.360,140.298,428.926,174.180,23.741,154.099
C07934=1078.354,140.049,428.947,174.179,23.738,154.099
C07935=1078.349,139.800,428.967,174.177,23.736,154.099
C07936=1078.343,139.551,428.987,174.175,23.734,154.099
C07937=1078.338,139.302,429.008,174.173,23.731,154.098
C07938=1078.332,139.053,429.028,174.171,23.729,154.098
C07939=1078.327,138.804,429.049,174.169,23.726,154.098
C07940=1078.320,138.554,429.069,174.167,23.724,154.098
C07941=1078.315,138.305,429.089,174.166,23.722,154.097
C07942=1078.309,138.056,429.110,174.163,23.720,154.097
C07943=1078.303,137.807,429.130,174.162,23.717,154.097
C07944=1078.298,137.558,429.150,174.159,23.715,154.097
C07945=1078.292,137.309,429.170,174.158,23.713,154.097
C07946=1078.287,137.060,429.191,174.156,23.711,154.096
C07947=1078.281,136.810,429.211,174.154,23.708,154.096
C07948=1078.275,136.561,429.231,174.152,23.706,154.096
C07949=1078.269,136.312,429.251,174.150,23.703,154.096
C07950=1078.263,136.063,429.271,174.148,23.701,154.095
C07951=1078.258,135.814,429.292,174.146,23.699,154.095
C07952=1078.252,135.566,429.312,174.145,23.696,154.095
C07953=1078.247,135.316,429.332,174.142,23.694,154.095
C07954=1078.241,135.067,429.351,174.141,23.692,154.095
C07955=1078.236,134.818,429.372,174.139,23.689,154.094
C07956=1078.230,134.569,429.392,174.137,23.687,154.094
C07957=1078.225,134.320,429.412,174.135,23.685,154.094
C07958=1078.218,134.070,429.433,174.134,23.682,154.094
C07959=1078.213,133.821,429.453,174.131,23.680,154.093
C07960=1078.207,133.572,429.473,174.130,23.678,154.093
C07961=1078.202,133.323,429.493,174.128,23.675,154.093
C07962=1078.196,133.074,429.513,174.126,23.673,154.093
C07963=1078.190,132.824,429.532,174.124,23.671,154.093
C07964=1078.185,132.575,429.553,174.122,23.668,154.092
C07965=1078.179,132.327,429.573,174.120,23.666,154.092
C07966=1078.174,132.077,429.593,174.118,23.663,154.092
C07967=1078.168,131.828,429.613,174.117,23.661,154.092
C07968=1078.162,131.579,429.633,174.114,23.659,154.091
C07969=1078.156,131.330,429.653,174.113,23.657,154.091
C07970=1078.151,131.081,429.672,174.111,23.654,154.091
C07971=1078.145,130.832,429.692,174.109,23.652,154.091
C07972=1078.139,130.583,429.712,174.107,23.649,154.091
C07973=1078.133,130.334,429.732,174.106,23.648,154.090
C07974=1078.128,130.084,429.752,174.103,23.645,154.090
C07975=1078.122,129.835,429.772,174.102,23.642,154.090
C07976=1078.116,129.585,429.792,174.100,23.640,154.090
C07977=1078.110,129.337,429.812,174.098,23.638,154.089
C07978=1078.104,129.088,429.832,174.096,23.636,154.089
C07979=1078.099,128.838,429.851,174.095,23.633,154.089
C07980=1078.093,128.589,429.871,174.092,23.631,154.089
C07981=1078.087,128.340,429.891,174.091,23.629,154.089
C07982=1078.081,128.091,429.911,174.089,23.626,154.088
C07983=1078.076,127.842,429.930,174.087,23.624,154.088
C07984=1078.069,127.561,429.952,174.085,23.621,154.088
C07985=1078.063,127.280,429.975,174.083,23.619,154.088
C07986=1078.057,126.999,429.997,174.081,23.616,154.087
C07987=1078.050,126.718,430.019,174.079,23.613,154.087
C07988=1078.044,126.469,430.039,174.077,23.611,154.087
C07989=1078.038,126.220,430.059,174.076,23.609,154.087
C07990=1078.033,125.970,430.078,174.073,23.607,154.087
C07991=1078.027,125.721,430.098,174.072,23.604,154.086
C07992=1078.022,125.472,430.118,174.070,23.602,154.086
C07993=1078.016,125.223,430.138,174.068,23.600,154.086
C07994=1078.010,124.974,430.156,174.066,23.597,154.086
C07995=1078.004,124.725,430.176,174.065,23.595,154.085
C07996=1077.999,124.476,430.196,174.062,23.592,154.085
C07997=1077.993,124.227,430.216,174.061,23.590,154.085
C07998=1077.988,123.977,430.235,174.059,23.588,154.085
C07999=1077.982,123.728,430.255,174.057,23.585,154.084
C08000=1077.976,123.479,430.275,174.055,23.583,154.084
C08001=1077.970,123.230,430.294,174.054,23.581,154.084
C08002=1077.964,122.981,430.314,174.052,23.578,154.084
C08003=1077.959,122.732,430.333,174.050,23.576,154.084
C08004=1077.953,122.482,430.352,174.048,23.573,154.083
C08005=1077.947,122.233,430.372,174.047,23.571,154.083
C08006=1077.942,121.985,430.391,174.044,23.569,154.083
C08007=1077.937,121.735,430.411,174.043,23.566,154.083
C08008=1077.931,121.486,430.431,174.041,23.564,154.082
C08009=1077.925,121.237,430.450,174.039,23.561,154.082
C08010=1077.920,120.987,430.469,174.038,23.559,154.082
C08011=1077.914,120.738,430.489,174.036,23.557,154.082
C08012=1077.908,120.489,430.509,174.034,23.554,154.081
C08013=1077.902,120.239,430.528,174.032,23.552,154.081
C08014=1077.897,119.991,430.547,174.031,23.550,154.081
C08015=1077.891,119.742,430.567,174.028,23.547,154.081
C08016=1077.886,119.492,430.586,174.027,23.545,154.080
C08017=1077.880,119.243,430.605,174.025,23.542,154.080
C08018=1077.874,118.994,430.625,174.023,23.540,154.080
C08019=1077.868,118.745,430.644,174.021,23.537,154.080
C08020=1077.864,118.496,430.664,174.020,23.535,154.079
C08021=1077.858,118.246,430.683,174.019,23.533,154.079
C08022=1077.852,117.997,430.702,174.016,23.530,154.079
C08023=1077.847,117.747,430.722,174.015,23.528,154.079
C08024=1077.841,117.499,430.742,174.013,23.526,154.078
C08025=1077.836,117.250,430.760,174.011,23.523,154.078
C08026=1077.830,117.000,430.780,174.009,23.520,154.078
C08027=1077.824,116.751,430.799,174.008,23.518,154.078
C08028=1077.819,116.502,430.818,174.005,23.516,154.077
C08029=1077.814,116.253,430.837,174.004,23.513,154.077
C08030=1077.808,116.004,430.857,174.003,23.511,154.077
C08031=1077.802,115.755,430.876,174.001,23.508,154.077
C08032=1077.796,115.505,430.896,173.999,23.506,154.076
C08033=1077.791,115.256,430.914,173.997,23.504,154.076
C08034=1077.785,115.007,430.934,173.996,23.501,154.076
C08035=1077.780,114.758,430.953,173.993,23.499,154.076
C08036=1077.774,114.508,430.972,173.992,23.496,154.075
C08037=1077.769,114.259,430.991,173.990,23.493,154.075
C08038=1077.763,114.010,431.010,173.988,23.492,154.075
C08039=1077.758,113.761,431.030,173.987,23.489,154.075
C08040=1077.751,113.511,431.048,173.985,23.486,154.074
C08041=1077.745,113.262,431.067,173.984,23.485,154.074
C08042=1077.740,113.013,431.086,173.981,23.482,154.074
C08043=1077.735,112.764,431.106,173.980,23.479,154.074
C08044=1077.729,112.514,431.125,173.978,23.477,154.073
C08045=1077.723,112.265,431.143,173.976,23.475,154.073
C08046=1077.717,112.017,431.162,173.975,23.472,154.073
C08047=1077.712,111.767,431.182,173.973,23.470,154.073
C08048=1077.705,111.486,431.203,173.971,23.467,154.072
C08049=1077.698,111.205,431.224,173.969,23.464,154.072
C08050=1077.692,110.924,431.246,173.967,23.462,154.072
C08051=1077.686,110.643,431.267,173.965,23.459,154.072
C08052=1077.680,110.394,431.286,173.964,23.457,154.071
C08053=1077.675,110.145,431.305,173.961,23.454,154.071
C08054=1077.669,109.896,431.324,173.960,23.452,154.071
C08055=1077.662,109.647,431.343,173.959,23.450,154.071
C08056=1077.657,109.397,431.362,173.956,23.447,154.070
C08057=1077.652,109.148,431.381,173.955,23.445,154.070
C08058=1077.645,108.899,431.400,173.953,23.442,154.070
C08059=1077.640,108.649,431.418,173.952,23.440,154.070
C08060=1077.634,108.400,431.437,173.950,23.438,154.069
C08061=1077.628,108.151,431.456,173.948,23.435,154.069
C08062=1077.623,107.902,431.475,173.947,23.433,154.069
C08063=1077.617,107.653,431.494,173.944,23.430,154.069
C08064=1077.611,107.404,431.512,173.943,23.428,154.068
C08065=1077.606,107.154,431.531,173.942,23.426,154.068
C08066=1077.600,106.905,431.550,173.939,23.423,154.068
C08067=1077.594,106.656,431.569,173.938,23.421,154.068
C08068=1077.589,106.407,431.588,173.936,23.418,154.067
C08069=1077.583,106.157,431.607,173.934,23.416,154.067
C08070=1077.577,105.908,431.625,173.933,23.414,154.067
C08071=1077.572,105.659,431.644,173.931,23.411,154.067
C08072=1077.566,105.409,431.663,173.930,23.408,154.066
C08073=1077.560,105.160,431.682,173.927,23.406,154.066
C08074=1077.555,104.911,431.700,173.926,23.404,154.066
C08075=1077.548,104.662,431.718,173.925,23.401,154.066
C08076=1077.543,104.413,431.737,173.923,23.399,154.065
C08077=1077.538,104.163,431.756,173.921,23.396,154.065
C08078=1077.531,103.914,431.775,173.919,23.394,154.065
C08079=1077.526,103.665,431.793,173.918,23.392,154.065
C08080=1077.520,103.416,431.812,173.916,23.389,154.064
C08081=1077.515,103.166,431.831,173.914,23.386,154.064
C08082=1077.509,102.917,431.849,173.913,23.384,154.064
C08083=1077.503,102.668,431.868,173.911,23.382,154.064
C08084=1077.498,102.419,431.886,173.909,23.379,154.063
C08085=1077.492,102.170,431.905,173.908,23.377,154.063
C08086=1077.486,101.920,431.923,173.906,23.374,154.063
C08087=1077.481,101.671,431.942,173.904,23.372,154.062
C08088=1077.475,101.422,431.961,173.903,23.369,154.062
C08089=1077.470,101.172,431.979,173.901,23.367,154.062
C08090=1077.464,100.923,431.998,173.899,23.365,154.062
C08091=1077.458,100.674,432.016,173.897,23.362,154.062
C08092=1077.453,100.425,432.035,173.896,23.360,154.061
C08093=1077.446,100.176,432.053,173.895,23.357,154.061
C08094=1077.441,99.926,432.072,173.892,23.355,154.061
C08095=1077.435,99.677,432.090,173.891,23.353,154.060
C08096=1077.429,99.428,432.108,173.890,23.350,154.060
C08097=1077.424,99.179,432.127,173.888,23.347,154.060
C08098=1077.418,98.929,432.145,173.886,23.346,154.060
C08099=1077.412,98.680,432.164,173.884,23.343,154.060
C08100=1077.406,98.431,432.182,173.883,23.340,154.059
C08101=1077.400,98.181,432.200,173.881,23.338,154.059
C08102=1077.395,97.932,432.218,173.879,23.335,154.059
C08103=1077.389,97.683,432.237,173.878,23.333,154.059
C08104=1077.383,97.434,432.255,173.876,23.331,154.058
C08105=1077.378,97.185,432.274,173.874,23.328,154.058
C08106=1077.371,96.935,432.292,173.873,23.326,154.058
C08107=1077.366,96.686,432.311,173.872,23.323,154.057
C08108=1077.360,96.436,432.329,173.869,23.321,154.057
C08109=1077.355,96.187,432.346,173.868,23.319,154.057
C08110=1077.349,95.938,432.365,173.867,23.316,154.057
C08111=1077.343,95.689,432.383,173.864,23.314,154.056
C08112=1077.336,95.408,432.404,173.862,23.311,154.056
C08113=1077.330,95.127,432.424,173.861,23.308,154.056
C08114=1077.324,94.847,432.445,173.859,23.305,154.055
C08115=1077.317,94.565,432.466,173.858,23.303,154.055
C08116=1077.312,94.316,432.483,173.855,23.300,154.055
C08117=1077.306,94.067,432.502,173.854,23.298,154.055
C08118=1077.301,93.817,432.520,173.852,23.295,154.054
C08119=1077.295,93.568,432.538,173.851,23.293,154.054
C08120=1077.289,93.319,432.557,173.849,23.291,154.054
C08121=1077.283,93.069,432.574,173.847,23.288,154.054
C08122=1077.278,92.820,432.593,173.846,23.285,154.053
C08123=1077.272,92.572,432.611,173.845,23.283,154.053
C08124=1077.266,92.322,432.629,173.842,23.280,154.053
C08125=1077.261,92.073,432.647,173.841,23.278,154.052
C08126=1077.255,91.823,432.665,173.840,23.275,154.052
C08127=1077.249,91.574,432.683,173.838,23.273,154.052
C08128=1077.244,91.324,432.702,173.836,23.270,154.052
C08129=1077.238,91.075,432.719,173.835,23.268,154.051
C08130=1077.232,90.826,432.737,173.833,23.266,154.051
C08131=1077.226,90.577,432.756,173.831,23.263,154.051
C08132=1077.220,90.327,432.773,173.830,23.261,154.051
C08133=1077.215,90.078,432.791,173.828,23.258,154.050
C08134=1077.209,89.829,432.809,173.827,23.256,154.050
C08135=1077.204,89.579,432.827,173.825,23.254,154.050
C08136=1077.197,89.330,432.846,173.823,23.251,154.050
C08137=1077.192,89.081,432.863,173.822,23.249,154.049
C08138=1077.186,88.831,432.881,173.820,23.246,154.049
C08139=1077.180,88.582,432.899,173.818,23.243,154.049
C08140=1077.174,88.333,432.917,173.817,23.241,154.049
C08141=1077.169,88.083,432.934,173.815,23.239,154.048
C08142=1077.163,87.835,432.953,173.813,23.236,154.048
C08143=1077.157,87.585,432.971,173.812,23.234,154.048
C08144=1077.151,87.336,432.988,173.811,23.232,154.048
C08145=1077.145,87.087,433.006,173.809,23.229,154.047
C08146=1077.140,86.838,433.024,173.807,23.226,154.047
C08147=1077.133,86.588,433.042,173.806,23.224,154.047
C08148=1077.128,86.339,433.059,173.804,23.221,154.046
C08149=1077.123,86.089,433.077,173.802,23.219,154.046
C08150=1077.117,85.840,433.095,173.801,23.217,154.046
C08151=1077.111,85.591,433.113,173.799,23.214,154.046
C08152=1077.105,85.341,433.131,173.798,23.212,154.045
C08153=1077.100,85.092,433.149,173.796,23.209,154.045
C08154=1077.094,84.843,433.167,173.794,23.206,154.045
C08155=1077.088,84.594,433.184,173.793,23.204,154.045
C08156=1077.082,84.345,433.202,173.792,23.202,154.044
C08157=1077.076,84.095,433.220,173.789,23.199,154.044
C08158=1077.071,83.846,433.238,173.788,23.196,154.044
C08159=1077.065,83.597,433.255,173.787,23.195,154.044
C08160=1077.059,83.347,433.273,173.785,23.192,154.043
C08161=1077.054,83.098,433.291,173.783,23.189,154.043
C08162=1077.048,82.849,433.308,173.782,23.187,154.043
C08163=1077.042,82.599,433.326,173.781,23.185,154.042
C08164=1077.036,82.350,433.344,173.779,23.182,154.042
C08165=1077.031,82.101,433.361,173.777,23.179,154.042
C08166=1077.025,81.851,433.378,173.776,23.177,154.042
C08167=1077.020,81.602,433.396,173.774,23.174,154.041
C08168=1077.014,81.353,433.414,173.772,23.172,154.041
C08169=1077.008,81.103,433.432,173.771,23.169,154.041
C08170=1077.002,80.854,433.449,173.769,23.167,154.040
C08171=1076.997,80.605,433.467,173.768,23.164,154.040
C08172=1076.991,80.355,433.485,173.766,23.162,154.040
C08173=1076.985,80.106,433.502,173.764,23.159,154.040
C08174=1076.980,79.857,433.520,173.763,23.157,154.039
C08175=1076.974,79.607,433.537,173.762,23.154,154.039
C08176=1076.967,79.326,433.556,173.760,23.151,154.039
C08177=1076.961,79.045,433.576,173.758,23.149,154.038
C08178=1076.954,78.764,433.596,173.756,23.146,154.038
C08179=1076.948,78.484,433.616,173.755,23.143,154.038
C08180=1076.942,78.235,433.633,173.753,23.140,154.038
C08181=1076.937,77.985,433.650,173.752,23.138,154.037
C08182=1076.931,77.736,433.668,173.750,23.136,154.037
C08183=1076.925,77.486,433.686,173.748,23.133,154.037
C08184=1076.919,77.238,433.703,173.747,23.130,154.036
C08185=1076.913,76.989,433.720,173.746,23.128,154.036
C08186=1076.908,76.738,433.738,173.743,23.125,154.036
C08187=1076.902,76.489,433.755,173.742,23.123,154.036
C08188=1076.897,76.240,433.773,173.741,23.121,154.035
C08189=1076.890,75.991,433.790,173.739,23.119,154.035
C08190=1076.884,75.741,433.807,173.737,23.116,154.035
C08191=1076.879,75.492,433.824,173.736,23.113,154.035
C08192=1076.873,75.243,433.842,173.735,23.111,154.034
C08193=1076.867,74.993,433.859,173.733,23.108,154.034
C08194=1076.861,74.744,433.876,173.731,23.106,154.034
C08195=1076.856,74.495,433.894,173.730,23.103,154.033
C08196=1076.850,74.246,433.911,173.729,23.101,154.033
C08197=1076.844,73.996,433.928,173.727,23.098,154.033
C08198=1076.838,73.747,433.946,173.725,23.096,154.033
C08199=1076.833,73.498,433.963,173.724,23.093,154.032
C08200=1076.828,73.248,433.980,173.722,23.091,154.032
C08201=1076.821,72.999,433.997,173.721,23.088,154.032
C08202=1076.815,72.749,434.014,173.719,23.086,154.031
C08203=1076.810,72.500,434.032,173.718,23.083,154.031
C08204=1076.804,72.251,434.049,173.716,23.081,154.031
C08205=1076.798,72.001,434.066,173.715,23.078,154.031
C08206=1076.792,71.752,434.083,173.713,23.076,154.030
C08207=1076.787,71.502,434.100,173.711,23.073,154.030
C08208=1076.781,71.253,434.117,173.710,23.070,154.030
C08209=1076.775,71.004,434.135,173.709,23.068,154.029
C08210=1076.770,70.754,434.152,173.707,23.066,154.029
C08211=1076.763,70.505,434.169,173.705,23.063,154.029
C08212=1076.758,70.256,434.186,173.704,23.060,154.029
C08213=1076.753,70.006,434.203,173.703,23.058,154.028
C08214=1076.747,69.757,434.220,173.700,23.056,154.028
C08215=1076.741,69.508,434.237,173.699,23.053,154.028
C08216=1076.735,69.258,434.254,173.698,23.051,154.028
C08217=1076.729,69.009,434.271,173.696,23.049,154.027
C08218=1076.724,68.759,434.288,173.694,23.046,154.027
C08219=1076.718,68.511,434.305,173.693,23.043,154.027
C08220=1076.712,68.261,434.322,173.692,23.041,154.026
C08221=1076.705,68.012,434.339,173.691,23.039,154.026
C08222=1076.700,67.762,434.356,173.688,23.036,154.026
C08223=1076.694,67.513,434.373,173.687,23.033,154.026
C08224=1076.689,67.263,434.390,173.686,23.031,154.025
C08225=1076.683,67.015,434.407,173.684,23.028,154.025
C08226=1076.677,66.765,434.424,173.682,23.026,154.025
C08227=1076.670,66.516,434.441,173.681,23.023,154.025
C08228=1076.665,66.266,434.458,173.680,23.021,154.024
C08229=1076.660,66.016,434.475,173.678,23.018,154.024
C08230=1076.654,65.768,434.492,173.676,23.016,154.024
C08231=1076.649,65.518,434.509,173.675,23.013,154.023
C08232=1076.642,65.269,434.526,173.674,23.011,154.023
C08233=1076.637,65.020,434.543,173.672,23.008,154.023
C08234=1076.631,64.770,434.559,173.670,23.006,154.023
C08235=1076.625,64.520,434.577,173.669,23.003,154.022
C08236=1076.619,64.271,434.593,173.668,23.001,154.022
C08237=1076.613,64.022,434.609,173.666,22.998,154.022
C08238=1076.608,63.773,434.627,173.665,22.996,154.021
C08239=1076.602,63.523,434.643,173.663,22.993,154.021
C08240=1076.595,63.242,434.662,173.661,22.990,154.021
C08241=1076.588,62.961,434.681,173.660,22.988,154.021
C08242=1076.581,62.680,434.700,173.658,22.985,154.020
C08243=1076.575,62.399,434.719,173.657,22.982,154.020
C08244=1076.569,62.150,434.735,173.654,22.979,154.020
C08245=1076.563,61.901,434.751,173.653,22.977,154.019
C08246=1076.557,61.651,434.769,173.652,22.975,154.019
C08247=1076.551,61.402,434.785,173.650,22.973,154.019
C08248=1076.545,61.152,434.802,173.648,22.970,154.019
C08249=1076.540,60.902,434.819,173.647,22.967,154.018
C08250=1076.533,60.654,434.836,173.646,22.965,154.018
C08251=1076.527,60.404,434.852,173.645,22.963,154.018
C08252=1076.521,60.155,434.868,173.642,22.960,154.018
C08253=1076.516,59.905,434.885,173.641,22.957,154.017
C08254=1076.510,59.656,434.901,173.640,22.955,154.017
C08255=1076.504,59.407,434.918,173.639,22.952,154.017
C08256=1076.498,59.158,434.934,173.636,22.950,154.016
C08257=1076.492,58.908,434.952,173.635,22.947,154.016
C08258=1076.486,58.658,434.968,173.634,22.945,154.016
C08259=1076.480,58.409,434.984,173.633,22.942,154.016
C08260=1076.474,58.160,435.001,173.630,22.940,154.015
C08261=1076.469,57.910,435.018,173.629,22.937,154.015
C08262=1076.463,57.661,435.034,173.628,22.935,154.015
C08263=1076.457,57.412,435.051,173.627,22.933,154.015
C08264=1076.451,57.162,435.067,173.624,22.930,154.014
C08265=1076.446,56.913,435.084,173.623,22.928,154.014
C08266=1076.440,56.663,435.100,173.622,22.925,154.014
C08267=1076.434,56.414,435.116,173.621,22.923,154.013
C08268=1076.428,56.165,435.132,173.618,22.920,154.013
C08269=1076.423,55.915,435.149,173.617,22.918,154.013
C08270=1076.416,55.666,435.166,173.616,22.915,154.013
C08271=1076.410,55.417,435.182,173.615,22.913,154.012
C08272=1076.405,55.168,435.199,173.612,22.910,154.012
C08273=1076.399,54.918,435.215,173.611,22.907,154.012
C08274=1076.393,54.669,435.232,173.610,22.905,154.011
C08275=1076.387,54.419,435.248,173.609,22.903,154.011
C08276=1076.381,54.170,435.264,173.607,22.900,154.011
C08277=1076.376,53.921,435.281,173.605,22.897,154.011
C08278=1076.370,53.671,435.297,173.604,22.895,154.010
C08279=1076.364,53.422,435.314,173.603,22.893,154.010
C08280=1076.358,53.172,435.330,173.601,22.890,154.010
C08281=1076.352,52.923,435.346,173.599,22.887,154.009
C08282=1076.347,52.674,435.362,173.598,22.885,154.009
C08283=1076.341,52.424,435.379,173.597,22.882,154.009
C08284=1076.335,52.175,435.395,173.596,22.880,154.008
C08285=1076.329,51.925,435.412,173.594,22.877,154.008
C08286=1076.323,51.676,435.428,173.592,22.874,154.008
C08287=1076.317,51.426,435.444,173.591,22.872,154.008
C08288=1076.312,51.177,435.460,173.590,22.869,154.007
C08289=1076.306,50.927,435.476,173.588,22.867,154.007
C08290=1076.300,50.678,435.492,173.586,22.864,154.007
C08291=1076.295,50.428,435.509,173.585,22.862,154.006
C08292=1076.289,50.179,435.526,173.584,22.859,154.006
C08293=1076.283,49.930,435.541,173.582,22.857,154.006
C08294=1076.277,49.681,435.558,173.581,22.854,154.006
C08295=1076.272,49.431,435.574,173.579,22.852,154.005
C08296=1076.266,49.182,435.590,173.578,22.849,154.005
C08297=1076.260,48.932,435.606,173.577,22.847,154.005
C08298=1076.255,48.682,435.623,173.575,22.844,154.005
C08299=1076.249,48.433,435.639,173.573,22.842,154.004
C08300=1076.243,48.184,435.655,173.572,22.839,154.004
C08301=1076.237,47.934,435.671,173.571,22.837,154.004
C08302=1076.232,47.686,435.687,173.569,22.834,154.003
C08303=1076.226,47.436,435.703,173.568,22.831,154.003
C08304=1076.219,47.155,435.722,173.566,22.829,154.003
C08305=1076.213,46.873,435.740,173.564,22.825,154.002
C08306=1076.207,46.592,435.758,173.563,22.823,154.002
C08307=1076.200,46.310,435.776,173.561,22.820,154.002
C08308=1076.194,46.061,435.792,173.560,22.817,154.001
C08309=1076.189,45.812,435.808,173.559,22.815,154.001
C08310=1076.183,45.563,435.824,173.557,22.812,154.001
C08311=1076.178,45.313,435.840,173.555,22.809,154.000
C08312=1076.172,45.064,435.856,173.554,22.807,154.000
C08313=1076.166,44.814,435.872,173.553,22.804,154.000
C08314=1076.160,44.565,435.889,173.552,22.802,154.000
C08315=1076.154,44.315,435.904,173.549,22.799,153.999
C08316=1076.149,44.067,435.920,173.548,22.797,153.999
C08317=1076.143,43.817,435.936,173.547,22.794,153.999
C08318=1076.137,43.567,435.952,173.546,22.791,153.998
C08319=1076.131,43.318,435.968,173.545,22.789,153.998
C08320=1076.125,43.069,435.984,173.542,22.786,153.998
C08321=1076.120,42.819,436.000,173.541,22.784,153.998
C08322=1076.114,42.570,436.016,173.540,22.781,153.997
C08323=1076.108,42.321,436.032,173.539,22.779,153.997
C08324=1076.103,42.071,436.048,173.537,22.776,153.997
C08325=1076.097,41.821,436.064,173.535,22.774,153.996
C08326=1076.091,41.571,436.079,173.534,22.771,153.996
C08327=1076.084,41.322,436.095,173.533,22.769,153.996
C08328=1076.079,41.074,436.111,173.532,22.766,153.996
C08329=1076.073,40.824,436.126,173.529,22.763,153.995
C08330=1076.067,40.574,436.143,173.528,22.761,153.995
C08331=1076.062,40.324,436.158,173.527,22.759,153.995
C08332=1076.056,40.075,436.175,173.526,22.756,153.994
C08333=1076.050,39.826,436.190,173.524,22.754,153.994
C08334=1076.045,39.576,436.206,173.522,22.751,153.994
C08335=1076.038,39.327,436.222,173.521,22.748,153.994
C08336=1076.032,39.077,436.237,173.520,22.746,153.993
C08337=1076.026,38.828,436.253,173.519,22.744,153.993
C08338=1076.021,38.579,436.269,173.517,22.741,153.993
C08339=1076.016,38.329,436.285,173.515,22.738,153.992
C08340=1076.010,38.079,436.300,173.514,22.736,153.992
C08341=1076.003,37.830,436.316,173.513,22.733,153.992
C08342=1075.998,37.581,436.331,173.511,22.731,153.992
C08343=1075.992,37.332,436.347,173.510,22.729,153.991
C08344=1075.987,37.082,436.363,173.508,22.726,153.991
C08345=1075.980,36.833,436.379,173.507,22.723,153.991
C08346=1075.974,36.583,436.394,173.506,22.721,153.990
C08347=1075.969,36.334,436.410,173.504,22.718,153.990
C08348=1075.962,36.084,436.425,173.503,22.716,153.990
C08349=1075.957,35.834,436.441,173.501,22.713,153.990
C08350=1075.951,35.585,436.457,173.500,22.711,153.989
C08351=1075.945,35.336,436.471,173.498,22.708,153.989
C08352=1075.939,35.087,436.488,173.497,22.706,153.989
C08353=1075.933,34.837,436.503,173.496,22.704,153.988
C08354=1075.927,34.588,436.519,173.494,22.701,153.988
C08355=1075.921,34.338,436.534,173.493,22.698,153.988
C08356=1075.916,34.089,436.550,173.491,22.696,153.988
C08357=1075.909,33.840,436.565,173.490,22.693,153.987
C08358=1075.904,33.590,436.581,173.489,22.691,153.987
C08359=1075.899,33.340,436.596,173.487,22.688,153.987
C08360=1075.892,33.091,436.612,173.485,22.686,153.986
C08361=1075.886,32.841,436.627,173.484,22.683,153.986
C08362=1075.881,32.591,436.643,173.483,22.681,153.986
C08363=1075.875,32.343,436.658,173.482,22.678,153.986
C08364=1075.869,32.093,436.674,173.480,22.676,153.985
C08365=1075.863,31.843,436.688,173.478,22.673,153.985
C08366=1075.857,31.595,436.704,173.477,22.671,153.985
C08367=1075.852,31.345,436.720,173.476,22.668,153.984
C08368=1075.845,31.063,436.737,173.474,22.665,153.984
C08369=1075.838,30.782,436.754,173.473,22.662,153.984
C08370=1075.832,30.502,436.771,173.471,22.660,153.984
C08371=1075.825,30.220,436.789,173.470,22.657,153.983
C08372=1075.819,29.970,436.804,173.468,22.654,153.983
C08373=1075.814,29.721,436.820,173.467,22.652,153.983
C08374=1075.808,29.472,436.836,173.465,22.649,153.982
C08375=1075.802,29.223,436.850,173.464,22.646,153.982
C08376=1075.796,28.973,436.866,173.462,22.644,153.982
C08377=1075.790,28.723,436.881,173.461,22.642,153.981
C08378=1075.785,28.474,436.896,173.460,22.639,153.981
C08379=1075.778,28.225,436.912,173.458,22.636,153.981
C08380=1075.773,27.975,436.927,173.457,22.634,153.981
C08381=1075.766,27.725,436.942,173.455,22.631,153.980
C08382=1075.761,27.476,436.957,173.454,22.630,153.980
C08383=1075.755,27.226,436.972,173.453,22.627,153.980
C08384=1075.750,26.977,436.988,173.451,22.624,153.980
C08385=1075.743,26.728,437.003,173.449,22.622,153.979
C08386=1075.737,26.478,437.019,173.448,22.619,153.979
C08387=1075.732,26.229,437.033,173.447,22.617,153.979
C08388=1075.725,25.979,437.048,173.446,22.615,153.978
C08389=1075.720,25.729,437.064,173.444,22.612,153.978
C08390=1075.714,25.480,437.078,173.442,22.609,153.978
C08391=1075.708,25.230,437.094,173.441,22.607,153.978
C08392=1075.702,24.981,437.109,173.440,22.604,153.977
C08393=1075.696,24.732,437.125,173.439,22.602,153.977
C08394=1075.690,24.482,437.140,173.437,22.599,153.977
C08395=1075.684,24.233,437.155,173.435,22.597,153.976
C08396=1075.679,23.983,437.170,173.434,22.594,153.976
C08397=1075.672,23.734,437.185,173.433,22.592,153.976
C08398=1075.667,23.485,437.200,173.431,22.589,153.976
C08399=1075.661,23.235,437.215,173.430,22.587,153.975
C08400=1075.654,22.985,437.230,173.429,22.584,153.975
C08401=1075.649,22.736,437.245,173.427,22.582,153.975
C08402=1075.643,22.486,437.260,173.426,22.579,153.974
C08403=1075.638,22.237,437.275,173.424,22.577,153.974
C08404=1075.632,21.987,437.290,173.423,22.574,153.974
C08405=1075.625,21.738,437.305,173.422,22.572,153.974
C08406=1075.620,21.488,437.320,173.420,22.569,153.973
C08407=1075.614,21.239,437.335,173.419,22.567,153.973
C08408=1075.608,20.990,437.350,173.417,22.564,153.973
C08409=1075.602,20.740,437.365,173.416,22.562,153.972
C08410=1075.597,20.491,437.380,173.415,22.559,153.972
C08411=1075.590,20.241,437.395,173.414,22.557,153.972
C08412=1075.585,19.992,437.410,173.411,22.554,153.972
C08413=1075.579,19.742,437.425,173.410,22.552,153.972
C08414=1075.573,19.492,437.439,173.409,22.550,153.971
C08415=1075.568,19.243,437.454,173.408,22.547,153.971
C08416=1075.561,18.993,437.469,173.406,22.545,153.971
C08417=1075.556,18.744,437.484,173.405,22.542,153.970
C08418=1075.549,18.495,437.499,173.403,22.539,153.970
C08419=1075.544,18.245,437.514,173.402,22.537,153.970
C08420=1075.538,17.996,437.529,173.401,22.535,153.970
C08421=1075.532,17.747,437.543,173.399,22.532,153.969
C08422=1075.526,17.497,437.558,173.398,22.530,153.969
C08423=1075.520,17.246,437.573,173.397,22.527,153.969
C08424=1075.514,16.997,437.588,173.395,22.524,153.968
C08425=1075.508,16.748,437.603,173.394,22.522,153.968
C08426=1075.502,16.499,437.617,173.392,22.519,153.968
C08427=1075.496,16.249,437.632,173.391,22.518,153.968
C08428=1075.491,16.000,437.647,173.390,22.515,153.967
C08429=1075.485,15.750,437.662,173.388,22.513,153.967
C08430=1075.479,15.501,437.676,173.386,22.510,153.967
C08431=1075.473,15.251,437.691,173.385,22.507,153.967
C08432=1075.467,14.971,437.708,173.384,22.504,153.966
C08433=1075.460,14.691,437.724,173.382,22.502,153.966
C08434=1075.453,14.412,437.741,173.381,22.499,153.966
C08435=1075.446,14.132,437.757,173.379,22.496,153.965
C08436=1075.441,13.882,437.772,173.377,22.494,153.965
C08437=1075.435,13.633,437.786,173.376,22.491,153.965
C08438=1075.429,13.383,437.801,173.375,22.489,153.964
C08439=1075.423,13.134,437.816,173.374,22.486,153.964
C08440=1075.417,12.884,437.831,173.372,22.484,153.964
C08441=1075.411,12.635,437.845,173.370,22.482,153.964
C08442=1075.405,12.385,437.860,173.369,22.479,153.963
C08443=1075.399,12.136,437.874,173.368,22.477,153.963
C08444=1075.393,11.886,437.888,173.366,22.474,153.963
C08445=1075.387,11.637,437.903,173.365,22.472,153.963
C08446=1075.381,11.387,437.918,173.364,22.469,153.962
C08447=1075.375,11.138,437.932,173.362,22.467,153.962
C08448=1075.369,10.888,437.947,173.360,22.465,153.962
C08449=1075.363,10.639,437.961,173.359,22.462,153.962
C08450=1075.357,10.389,437.976,173.358,22.460,153.961
C08451=1075.351,10.140,437.990,173.357,22.457,153.961
C08452=1075.345,9.890,438.005,173.356,22.455,153.961
C08453=1075.340,9.641,438.019,173.353,22.452,153.961
C08454=1075.333,9.391,438.034,173.352,22.450,153.960
C08455=1075.328,9.142,438.048,173.351,22.448,153.960
C08456=1075.321,8.892,438.063,173.350,22.445,153.960
C08457=1075.316,8.643,438.077,173.348,22.443,153.959
C08458=1075.310,8.393,438.091,173.347,22.440,153.959
C08459=1075.304,8.144,438.106,173.346,22.438,153.959
C08460=1075.298,7.894,438.120,173.344,22.435,153.959
C08461=1075.292,7.644,438.135,173.342,22.433,153.958
C08462=1075.286,7.395,438.149,173.341,22.431,153.958
C08463=1075.280,7.146,438.163,173.340,22.428,153.958
C08464=1075.274,6.896,438.177,173.339,22.426,153.958
C08465=1075.268,6.647,438.192,173.337,22.423,153.957
C08466=1075.262,6.397,438.206,173.335,22.420,153.957
C08467=1075.256,6.148,438.220,173.334,22.418,153.957
C08468=1075.251,5.898,438.234,173.333,22.416,153.957
C08469=1075.244,5.649,438.249,173.332,22.414,153.956
C08470=1075.239,5.399,438.263,173.330,22.411,153.956
C08471=1075.232,5.149,438.278,173.329,22.409,153.956
C08472=1075.227,4.900,438.292,173.327,22.406,153.956
C08473=1075.221,4.651,438.306,173.326,22.403,153.955
C08474=1075.215,4.400,438.321,173.325,22.401,153.955
C08475=1075.209,4.152,438.335,173.323,22.399,153.955
C08476=1075.204,3.902,438.349,173.322,22.397,153.954
C08477=1075.197,3.652,438.364,173.321,22.394,153.954
C08478=1075.192,3.403,438.378,173.319,22.392,153.954
C08479=1075.186,3.153,438.391,173.317,22.389,153.954
C08480=1075.179,2.904,438.406,173.316,22.386,153.953
C08481=1075.174,2.654,438.420,173.315,22.384,153.953
C08482=1075.168,2.405,438.435,173.313,22.382,153.953
C08483=1075.162,2.155,438.449,173.312,22.380,153.953
C08484=1075.157,1.905,438.463,173.311,22.377,153.952
C08485=1075.151,1.656,438.477,173.309,22.374,153.952
C08486=1075.145,1.406,438.491,173.308,22.372,153.952
C08487=1075.139,1.157,438.505,173.306,22.369,153.952
C08488=1075.133,0.908,438.520,173.305,22.367,153.951
C08489=1075.127,0.658,438.534,173.304,22.365,153.951
C08490=1075.121,0.409,438.548,173.303,22.363,153.951
C08491=1075.115,0.159,438.562,173.301,22.360,153.950
C08492=1075.110,-0.090,438.576,173.299,22.357,153.950
C08493=1075.104,-0.341,438.590,173.298,22.355,153.950
C08494=1075.098,-0.590,438.605,173.297,22.352,153.950
C08495=1075.093,-0.839,438.619,173.296,22.350,153.949
C08496=1075.085,-1.117,438.634,173.294,22.347,153.949
C08497=1075.079,-1.395,438.650,173.292,22.345,153.949
C08498=1075.073,-1.672,438.666,173.291,22.342,153.949
C08499=1075.066,-1.951,438.681,173.289,22.339,153.948
C08500=1075.061,-2.200,438.696,173.288,22.337,153.948
C08501=1075.054,-2.449,438.709,173.287,22.334,153.948
C08502=1075.049,-2.699,438.723,173.285,22.332,153.947
C08503=1075.043,-2.949,438.737,173.284,22.329,153.947
C08504=1075.037,-3.198,438.752,173.283,22.327,153.947
C08505=1075.032,-3.448,438.765,173.281,22.325,153.947
C08506=1075.025,-3.697,438.779,173.279,22.322,153.946
C08507=1075.019,-3.947,438.793,173.278,22.320,153.946
C08508=1075.014,-4.197,438.807,173.277,22.318,153.946
C08509=1075.007,-4.446,438.821,173.276,22.315,153.946
C08510=1075.001,-4.696,438.835,173.274,22.313,153.945
C08511=1074.995,-4.945,438.848,173.273,22.310,153.945
C08512=1074.990,-5.195,438.862,173.271,22.308,153.945
C08513=1074.984,-5.444,438.876,173.270,22.306,153.945
C08514=1074.977,-5.694,438.890,173.268,22.303,153.944
C08515=1074.972,-5.943,438.904,173.267,22.301,153.944
C08516=1074.965,-6.192,438.917,173.266,22.299,153.944
C08517=1074.959,-6.443,438.932,173.265,22.296,153.944
C08518=1074.954,-6.692,438.946,173.263,22.294,153.943
C08519=1074.948,-6.942,438.959,173.261,22.292,153.943
C08520=1074.942,-7.191,438.973,173.260,22.289,153.943
C08521=1074.935,-7.441,438.986,173.259,22.287,153.943
C08522=1074.930,-7.691,439.000,173.257,22.285,153.943
C08523=1074.924,-7.940,439.014,173.256,22.282,153.942
C08524=1074.918,-8.189,439.028,173.255,22.280,153.942
C08525=1074.912,-8.438,439.042,173.254,22.277,153.942
C08526=1074.905,-8.688,439.056,173.251,22.275,153.942
C08527=1074.900,-8.938,439.069,173.250,22.273,153.941
C08528=1074.894,-9.187,439.083,173.249,22.270,153.941
C08529=1074.888,-9.437,439.097,173.248,22.268,153.941
C08530=1074.883,-9.686,439.110,173.246,22.266,153.941
C08531=1074.876,-9.936,439.124,173.245,22.263,153.940
C08532=1074.871,-10.186,439.138,173.244,22.261,153.940
C08533=1074.864,-10.435,439.151,173.242,22.259,153.940
C08534=1074.859,-10.685,439.165,173.240,22.256,153.940
C08535=1074.853,-10.934,439.178,173.239,22.254,153.939
C08536=1074.847,-11.184,439.192,173.238,22.252,153.939
C08537=1074.840,-11.434,439.206,173.237,22.249,153.939
C08538=1074.835,-11.683,439.220,173.235,22.247,153.939
C08539=1074.829,-11.932,439.233,173.234,22.245,153.938
C08540=1074.823,-12.182,439.247,173.232,22.242,153.938
C08541=1074.817,-12.431,439.260,173.231,22.240,153.938
C08542=1074.812,-12.681,439.273,173.229,22.238,153.938
C08543=1074.805,-12.931,439.287,173.228,22.235,153.937
C08544=1074.799,-13.181,439.301,173.227,22.233,153.937
C08545=1074.794,-13.431,439.315,173.226,22.230,153.937
C08546=1074.788,-13.680,439.328,173.224,22.228,153.937
C08547=1074.782,-13.929,439.342,173.222,22.225,153.936
C08548=1074.776,-14.179,439.355,173.221,22.223,153.936
C08549=1074.771,-14.428,439.369,173.220,22.221,153.936
C08550=1074.764,-14.678,439.382,173.218,22.219,153.936
C08551=1074.759,-14.927,439.396,173.217,22.216,153.935
C08552=1074.752,-15.178,439.409,173.216,22.214,153.935
C08553=1074.746,-15.427,439.422,173.214,22.212,153.935
C08554=1074.741,-15.677,439.436,173.213,22.210,153.935
C08555=1074.735,-15.926,439.449,173.211,22.207,153.935
C08556=1074.728,-16.175,439.463,173.210,22.205,153.934
C08557=1074.723,-16.425,439.476,173.208,22.203,153.934
C08558=1074.717,-16.675,439.489,173.207,22.200,153.934
C08559=1074.710,-16.924,439.503,173.206,22.198,153.934
C08560=1074.703,-17.200,439.518,173.204,22.195,153.933
C08561=1074.697,-17.477,439.532,173.202,22.193,153.933
C08562=1074.691,-17.753,439.547,173.201,22.190,153.933
C08563=1074.685,-18.029,439.562,173.199,22.188,153.933
C08564=1074.678,-18.279,439.575,173.198,22.186,153.932
C08565=1074.672,-18.528,439.589,173.197,22.183,153.932
C08566=1074.665,-18.777,439.602,173.195,22.181,153.932
C08567=1074.660,-19.028,439.615,173.194,22.179,153.932
C08568=1074.654,-19.277,439.628,173.193,22.176,153.931
C08569=1074.648,-19.526,439.642,173.191,22.174,153.931
C08570=1074.642,-19.776,439.655,173.189,22.172,153.931
C08571=1074.636,-20.026,439.668,173.188,22.170,153.931
C08572=1074.630,-20.275,439.681,173.187,22.167,153.931
C08573=1074.624,-20.524,439.694,173.185,22.165,153.930
C08574=1074.619,-20.774,439.708,173.184,22.163,153.930
C08575=1074.613,-21.024,439.721,173.183,22.160,153.930
C08576=1074.606,-21.273,439.734,173.181,22.158,153.930
C08577=1074.601,-21.524,439.748,173.180,22.156,153.929
C08578=1074.594,-21.773,439.761,173.178,22.154,153.929
C08579=1074.588,-22.022,439.774,173.177,22.151,153.929
C08580=1074.582,-22.272,439.787,173.175,22.149,153.929
C08581=1074.577,-22.522,439.801,173.174,22.147,153.929
C08582=1074.571,-22.771,439.814,173.173,22.145,153.928
C08583=1074.565,-23.021,439.826,173.172,22.142,153.928
C08584=1074.558,-23.270,439.840,173.170,22.140,153.928
C08585=1074.553,-23.520,439.854,173.169,22.138,153.928
C08586=1074.547,-23.770,439.866,173.167,22.135,153.927
C08587=1074.541,-24.019,439.879,173.166,22.133,153.927
C08588=1074.535,-24.269,439.892,173.164,22.131,153.927
C08589=1074.530,-24.518,439.906,173.163,22.129,153.927
C08590=1074.524,-24.768,439.918,173.162,22.126,153.927
C08591=1074.517,-25.018,439.932,173.160,22.124,153.926
C08592=1074.511,-25.267,439.945,173.159,22.122,153.926
C08593=1074.505,-25.517,439.957,173.158,22.120,153.926
C08594=1074.500,-25.766,439.971,173.156,22.117,153.926
C08595=1074.494,-26.016,439.984,173.154,22.115,153.926
C08596=1074.488,-26.265,439.997,173.153,22.113,153.925
C08597=1074.482,-26.515,440.009,173.152,22.111,153.925
C08598=1074.476,-26.764,440.023,173.150,22.108,153.925
C08599=1074.471,-27.014,440.036,173.149,22.106,153.925
C08600=1074.465,-27.263,440.049,173.148,22.104,153.924
C08601=1074.459,-27.513,440.062,173.146,22.102,153.924
C08602=1074.453,-27.762,440.075,173.144,22.099,153.924
C08603=1074.447,-28.012,440.087,173.143,22.097,153.924
C08604=1074.441,-28.262,440.101,173.142,22.095,153.924
C08605=1074.435,-28.511,440.113,173.140,22.093,153.923
C08606=1074.428,-28.761,440.127,173.139,22.091,153.923
C08607=1074.422,-29.011,440.139,173.138,22.088,153.923
C08608=1074.417,-29.260,440.152,173.136,22.086,153.923
C08609=1074.410,-29.510,440.165,173.135,22.085,153.923
C08610=1074.404,-29.760,440.177,173.133,22.082,153.922
C08611=1074.398,-30.009,440.191,173.132,22.080,153.922
C08612=1074.392,-30.259,440.203,173.130,22.077,153.922
C08613=1074.386,-30.508,440.217,173.129,22.075,153.922
C08614=1074.380,-30.758,440.229,173.128,22.073,153.922
C08615=1074.374,-31.008,440.242,173.126,22.071,153.921
C08616=1074.368,-31.257,440.255,173.125,22.069,153.921
C08617=1074.362,-31.507,440.267,173.124,22.067,153.921
C08618=1074.356,-31.757,440.280,173.122,22.065,153.921
C08619=1074.350,-32.006,440.293,173.120,22.062,153.921
C08620=1074.344,-32.256,440.306,173.119,22.060,153.920
C08621=1074.338,-32.506,440.318,173.118,22.058,153.920
C08622=1074.333,-32.754,440.331,173.116,22.055,153.920
C08623=1074.327,-33.004,440.344,173.115,22.054,153.920
C08624=1074.319,-33.280,440.358,173.114,22.052,153.920
C08625=1074.313,-33.555,440.373,173.111,22.049,153.919
C08626=1074.306,-33.831,440.386,173.110,22.046,153.919
C08627=1074.299,-34.106,440.400,173.109,22.044,153.919
C08628=1074.294,-34.356,440.412,173.108,22.042,153.919
C08629=1074.287,-34.605,440.426,173.105,22.039,153.919
C08630=1074.282,-34.854,440.438,173.104,22.038,153.918
C08631=1074.276,-35.104,440.450,173.103,22.035,153.918
C08632=1074.270,-35.354,440.464,173.101,22.033,153.918
C08633=1074.264,-35.603,440.476,173.100,22.031,153.918
C08634=1074.258,-35.853,440.489,173.099,22.029,153.917
C08635=1074.252,-36.103,440.501,173.097,22.027,153.917
C08636=1074.246,-36.353,440.514,173.096,22.025,153.917
C08637=1074.241,-36.602,440.527,173.094,22.022,153.917
C08638=1074.235,-36.852,440.539,173.093,22.020,153.917
C08639=1074.229,-37.101,440.552,173.091,22.018,153.917
C08640=1074.223,-37.351,440.564,173.090,22.016,153.916
C08641=1074.216,-37.600,440.577,173.089,22.014,153.916
C08642=1074.210,-37.850,440.590,173.087,22.011,153.916
C08643=1074.205,-38.099,440.602,173.086,22.009,153.916
C08644=1074.199,-38.349,440.614,173.085,22.007,153.916
C08645=1074.193,-38.599,440.627,173.083,22.006,153.915
C08646=1074.187,-38.849,440.639,173.082,22.003,153.915
C08647=1074.181,-39.099,440.652,173.080,22.001,153.915
C08648=1074.174,-39.348,440.665,173.078,21.999,153.915
C08649=1074.169,-39.597,440.677,173.077,21.997,153.915
C08650=1074.163,-39.847,440.689,173.076,21.994,153.914
C08651=1074.157,-40.097,440.702,173.074,21.992,153.914
C08652=1074.150,-40.346,440.714,173.073,21.990,153.914
C08653=1074.145,-40.596,440.726,173.072,21.989,153.914
C08654=1074.139,-40.846,440.739,173.070,21.987,153.914
C08655=1074.133,-41.095,440.751,173.069,21.984,153.914
C08656=1074.127,-41.345,440.763,173.067,21.982,153.913
C08657=1074.120,-41.594,440.776,173.065,21.980,153.913
C08658=1074.115,-41.844,440.789,173.064,21.978,153.913
C08659=1074.108,-42.094,440.801,173.063,21.976,153.913
C08660=1074.103,-42.343,440.813,173.061,21.974,153.913
C08661=1074.097,-42.593,440.826,173.060,21.972,153.913
C08662=1074.090,-42.842,440.838,173.059,21.970,153.912
C08663=1074.084,-43.092,440.850,173.057,21.968,153.912
C08664=1074.078,-43.342,440.863,173.056,21.966,153.912
C08665=1074.073,-43.591,440.875,173.055,21.964,153.912
C08666=1074.066,-43.841,440.887,173.052,21.961,153.912
C08667=1074.060,-44.091,440.899,173.051,21.959,153.912
C08668=1074.054,-44.341,440.912,173.050,21.957,153.911
C08669=1074.048,-44.590,440.924,173.048,21.955,153.911
C08670=1074.043,-44.839,440.936,173.047,21.953,153.911
C08671=1074.037,-45.089,440.949,173.046,21.951,153.911
C08672=1074.030,-45.339,440.961,173.044,21.949,153.911
C08673=1074.024,-45.589,440.973,173.043,21.947,153.910
C08674=1074.019,-45.838,440.985,173.042,21.945,153.910
C08675=1074.012,-46.087,440.997,173.040,21.943,153.910
C08676=1074.006,-46.337,441.010,173.038,21.941,153.910
C08677=1074.001,-46.586,441.022,173.037,21.939,153.910
C08678=1073.995,-46.837,441.033,173.035,21.937,153.910
C08679=1073.989,-47.087,441.046,173.034,21.934,153.909
C08680=1073.983,-47.336,441.058,173.033,21.932,153.909
C08681=1073.977,-47.585,441.070,173.031,21.931,153.909
C08682=1073.971,-47.835,441.083,173.030,21.929,153.909
C08683=1073.965,-48.085,441.095,173.028,21.927,153.909
C08684=1073.959,-48.334,441.107,173.027,21.925,153.909
C08685=1073.953,-48.584,441.119,173.026,21.923,153.909
C08686=1073.946,-48.833,441.131,173.024,21.921,153.908
C08687=1073.941,-49.083,441.143,173.022,21.918,153.908
C08688=1073.934,-49.359,441.157,173.021,21.916,153.908
C08689=1073.927,-49.635,441.170,173.019,21.914,153.908
C08690=1073.921,-49.911,441.184,173.018,21.912,153.908
C08691=1073.915,-50.187,441.196,173.016,21.909,153.907
C08692=1073.908,-50.436,441.208,173.015,21.907,153.907
C08693=1073.903,-50.686,441.221,173.013,21.905,153.907
C08694=1073.896,-50.935,441.233,173.012,21.903,153.907
C08695=1073.890,-51.185,441.245,173.010,21.902,153.907
C08696=1073.884,-51.435,441.256,173.009,21.900,153.907
C08697=1073.878,-51.684,441.268,173.008,21.898,153.906
C08698=1073.872,-51.934,441.281,173.006,21.896,153.906
C08699=1073.866,-52.184,441.292,173.005,21.894,153.906
C08700=1073.859,-52.433,441.304,173.002,21.892,153.906
C08701=1073.854,-52.683,441.316,173.001,21.890,153.906
C08702=1073.847,-52.932,441.328,173.000,21.888,153.906
C08703=1073.841,-53.182,441.340,172.998,21.886,153.906
C08704=1073.835,-53.431,441.352,172.997,21.884,153.906
C08705=1073.829,-53.681,441.363,172.996,21.882,153.905
C08706=1073.822,-53.931,441.375,172.994,21.880,153.905
C08707=1073.817,-54.180,441.387,172.993,21.878,153.905
C08708=1073.811,-54.430,441.399,172.991,21.877,153.905
C08709=1073.804,-54.680,441.411,172.990,21.875,153.905
C08710=1073.798,-54.930,441.423,172.988,21.873,153.905
C08711=1073.792,-55.179,441.434,172.987,21.871,153.905
C08712=1073.786,-55.429,441.446,172.985,21.869,153.905
C08713=1073.780,-55.679,441.459,172.983,21.867,153.904
C08714=1073.774,-55.928,441.469,172.982,21.865,153.904
C08715=1073.767,-56.178,441.481,172.981,21.863,153.904
C08716=1073.761,-56.428,441.494,172.979,21.861,153.904
C08717=1073.756,-56.677,441.505,172.978,21.859,153.904
C08718=1073.749,-56.927,441.517,172.976,21.858,153.904
C08719=1073.744,-57.176,441.529,172.975,21.856,153.904
C08720=1073.737,-57.426,441.540,172.974,21.854,153.903
C08721=1073.731,-57.676,441.552,172.972,21.852,153.903
C08722=1073.725,-57.925,441.563,172.971,21.850,153.903
C08723=1073.719,-58.175,441.576,172.969,21.848,153.903
C08724=1073.713,-58.425,441.588,172.968,21.846,153.903
C08725=1073.707,-58.674,441.598,172.966,21.844,153.903
C08726=1073.701,-58.924,441.611,172.964,21.843,153.903
C08727=1073.695,-59.174,441.622,172.963,21.841,153.903
C08728=1073.688,-59.423,441.634,172.961,21.839,153.902
C08729=1073.682,-59.673,441.645,172.960,21.837,153.902
C08730=1073.677,-59.922,441.657,172.959,21.835,153.902
C08731=1073.670,-60.173,441.669,172.957,21.833,153.902
C08732=1073.664,-60.422,441.680,172.956,21.831,153.902
C08733=1073.659,-60.671,441.693,172.954,21.830,153.902
C08734=1073.653,-60.921,441.704,172.953,21.828,153.902
C08735=1073.646,-61.170,441.716,172.952,21.826,153.901
C08736=1073.640,-61.421,441.727,172.950,21.824,153.901
C08737=1073.634,-61.670,441.739,172.949,21.822,153.901
C08738=1073.628,-61.920,441.750,172.947,21.820,153.901
C08739=1073.622,-62.170,441.761,172.945,21.818,153.901
C08740=1073.616,-62.419,441.773,172.944,21.816,153.901
C08741=1073.611,-62.669,441.784,172.942,21.815,153.901
C08742=1073.604,-62.918,441.796,172.941,21.813,153.901
C08743=1073.598,-63.168,441.807,172.939,21.811,153.901
C08744=1073.592,-63.418,441.819,172.938,21.809,153.900
C08745=1073.586,-63.667,441.830,172.936,21.807,153.900
C08746=1073.580,-63.917,441.843,172.935,21.806,153.900
C08747=1073.574,-64.167,441.854,172.934,21.804,153.900
C08748=1073.568,-64.417,441.865,172.932,21.802,153.900
C08749=1073.561,-64.666,441.877,172.931,21.800,153.900
C08750=1073.556,-64.916,441.888,172.929,21.798,153.900
C08751=1073.550,-65.166,441.900,172.928,21.796,153.900
C08752=1073.544,-65.442,441.912,172.926,21.794,153.899
C08753=1073.537,-65.719,441.925,172.924,21.792,153.899
C08754=1073.530,-65.997,441.937,172.923,21.790,153.899
C08755=1073.523,-66.273,441.951,172.922,21.788,153.899
C08756=1073.517,-66.523,441.961,172.920,21.787,153.899
C08757=1073.512,-66.773,441.973,172.918,21.784,153.899
C08758=1073.506,-67.022,441.985,172.916,21.783,153.899
C08759=1073.499,-67.273,441.996,172.915,21.781,153.899
C08760=1073.494,-67.522,442.007,172.913,21.779,153.899
C08761=1073.487,-67.772,442.019,172.912,21.777,153.898
C08762=1073.482,-68.021,442.030,172.911,21.775,153.898
C08763=1073.476,-68.272,442.042,172.909,21.774,153.898
C08764=1073.470,-68.520,442.053,172.908,21.772,153.898
C08765=1073.464,-68.770,442.064,172.906,21.770,153.898
C08766=1073.457,-69.020,442.075,172.905,21.769,153.898
C08767=1073.452,-69.270,442.086,172.903,21.767,153.898
C08768=1073.446,-69.520,442.099,172.902,21.765,153.898
C08769=1073.440,-69.769,442.110,172.900,21.763,153.898
C08770=1073.434,-70.019,442.121,172.899,21.761,153.897
C08771=1073.428,-70.269,442.132,172.898,21.760,153.897
C08772=1073.422,-70.518,442.143,172.896,21.758,153.897
C08773=1073.416,-70.768,442.155,172.895,21.756,153.897
C08774=1073.411,-71.018,442.166,172.893,21.754,153.897
C08775=1073.405,-71.267,442.177,172.892,21.753,153.897
C08776=1073.398,-71.517,442.189,172.890,21.750,153.897
C08777=1073.392,-71.766,442.200,172.888,21.749,153.897
C08778=1073.386,-72.016,442.211,172.887,21.747,153.897
C08779=1073.380,-72.266,442.222,172.885,21.745,153.897
C08780=1073.375,-72.515,442.233,172.884,21.743,153.896
C08781=1073.369,-72.766,442.245,172.882,21.742,153.896
C08782=1073.363,-73.015,442.256,172.881,21.740,153.896
C08783=1073.357,-73.264,442.267,172.879,21.739,153.896
C08784=1073.351,-73.514,442.278,172.878,21.737,153.896
C08785=1073.345,-73.764,442.289,172.877,21.735,153.896
C08786=1073.339,-74.013,442.300,172.875,21.733,153.896
C08787=1073.333,-74.263,442.311,172.874,21.731,153.896
C08788=1073.327,-74.513,442.322,172.872,21.730,153.896
C08789=1073.321,-74.763,442.334,172.871,21.728,153.896
C08790=1073.315,-75.012,442.345,172.869,21.727,153.896
C08791=1073.309,-75.262,442.356,172.868,21.725,153.895
C08792=1073.303,-75.512,442.367,172.866,21.723,153.895
C08793=1073.297,-75.761,442.378,172.865,21.721,153.895
C08794=1073.290,-76.011,442.389,172.863,21.720,153.895
C08795=1073.284,-76.261,442.400,172.862,21.718,153.895
C08796=1073.279,-76.510,442.410,172.860,21.717,153.895
C08797=1073.272,-76.760,442.422,172.859,21.715,153.895
C08798=1073.267,-77.010,442.433,172.857,21.713,153.895
C08799=1073.261,-77.259,442.443,172.856,21.712,153.895
C08800=1073.254,-77.509,442.455,172.854,21.710,153.895
C08801=1073.249,-77.759,442.466,172.853,21.709,153.895
C08802=1073.242,-78.009,442.477,172.851,21.706,153.895
C08803=1073.237,-78.259,442.488,172.849,21.705,153.895
C08804=1073.230,-78.507,442.499,172.847,21.703,153.894
C08805=1073.223,-78.757,442.510,172.846,21.701,153.894
C08806=1073.218,-79.007,442.521,172.844,21.700,153.894
C08807=1073.212,-79.257,442.531,172.843,21.698,153.894
C08808=1073.207,-79.506,442.542,172.842,21.697,153.894
C08809=1073.200,-79.757,442.553,172.840,21.695,153.894
C08810=1073.194,-80.006,442.564,172.839,21.693,153.894
C08811=1073.187,-80.256,442.575,172.837,21.692,153.894
C08812=1073.182,-80.505,442.586,172.835,21.691,153.894
C08813=1073.176,-80.755,442.596,172.834,21.689,153.894
C08814=1073.169,-81.005,442.607,172.832,21.687,153.894
C08815=1073.163,-81.254,442.618,172.831,21.686,153.894
C08816=1073.156,-81.533,442.630,172.830,21.684,153.894
C08817=1073.149,-81.813,442.642,172.828,21.683,153.894
C08818=1073.142,-82.092,442.655,172.826,21.681,153.894
C08819=1073.136,-82.371,442.666,172.824,21.679,153.893
C08820=1073.129,-82.621,442.677,172.823,21.677,153.893
C08821=1073.123,-82.871,442.688,172.821,21.676,153.893
C08822=1073.117,-83.120,442.698,172.820,21.674,153.893
C08823=1073.111,-83.370,442.710,172.818,21.673,153.893
C08824=1073.104,-83.619,442.720,172.817,21.671,153.893
C08825=1073.099,-83.870,442.730,172.815,21.670,153.893
C08826=1073.093,-84.119,442.741,172.813,21.668,153.893
C08827=1073.086,-84.369,442.752,172.812,21.667,153.893
C08828=1073.080,-84.618,442.762,172.810,21.665,153.893
C08829=1073.075,-84.868,442.773,172.809,21.664,153.893
C08830=1073.068,-85.118,442.784,172.807,21.662,153.893
C08831=1073.062,-85.368,442.794,172.806,21.661,153.893
C08832=1073.056,-85.617,442.805,172.804,21.659,153.893
C08833=1073.049,-85.867,442.816,172.803,21.658,153.893
C08834=1073.044,-86.117,442.827,172.801,21.656,153.893
C08835=1073.038,-86.366,442.837,172.800,21.655,153.893
C08836=1073.032,-86.616,442.847,172.798,21.653,153.893
C08837=1073.025,-86.866,442.858,172.797,21.651,153.893
C08838=1073.020,-87.116,442.869,172.795,21.650,153.893
C08839=1073.013,-87.365,442.879,172.794,21.649,153.893
C08840=1073.008,-87.615,442.890,172.792,21.647,153.893
C08841=1073.001,-87.865,442.900,172.790,21.646,153.893
C08842=1072.995,-88.114,442.911,172.789,21.645,153.893
C08843=1072.989,-88.364,442.922,172.787,21.643,153.892
C08844=1072.983,-88.614,442.932,172.786,21.641,153.892
C08845=1072.977,-88.864,442.943,172.784,21.640,153.892
C08846=1072.970,-89.113,442.953,172.783,21.638,153.892
C08847=1072.964,-89.363,442.964,172.781,21.637,153.892
C08848=1072.959,-89.613,442.974,172.780,21.636,153.892
C08849=1072.952,-89.862,442.984,172.778,21.634,153.892
C08850=1072.946,-90.112,442.996,172.777,21.633,153.892
C08851=1072.940,-90.362,443.005,172.775,21.631,153.892
C08852=1072.934,-90.611,443.016,172.773,21.630,153.892
C08853=1072.928,-90.861,443.027,172.772,21.628,153.892
C08854=1072.922,-91.111,443.037,172.770,21.627,153.892
C08855=1072.916,-91.361,443.048,172.769,21.625,153.892
C08856=1072.909,-91.610,443.058,172.767,21.624,153.892
C08857=1072.904,-91.860,443.068,172.766,21.622,153.892
C08858=1072.898,-92.110,443.079,172.764,21.621,153.892
C08859=1072.892,-92.359,443.089,172.763,21.620,153.892
C08860=1072.886,-92.609,443.100,172.761,21.618,153.892
C08861=1072.879,-92.859,443.110,172.759,21.617,153.892
C08862=1072.874,-93.109,443.120,172.758,21.616,153.892
C08863=1072.867,-93.358,443.131,172.756,21.614,153.892
C08864=1072.862,-93.608,443.141,172.755,21.613,153.892
C08865=1072.856,-93.858,443.152,172.753,21.611,153.892
C08866=1072.850,-94.107,443.162,172.752,21.610,153.892
C08867=1072.844,-94.357,443.172,172.750,21.609,153.892
C08868=1072.837,-94.607,443.183,172.748,21.607,153.892
C08869=1072.832,-94.857,443.193,172.747,21.606,153.892
C08870=1072.825,-95.106,443.203,172.745,21.604,153.892
C08871=1072.820,-95.356,443.213,172.744,21.603,153.892
C08872=1072.813,-95.605,443.224,172.742,21.602,153.892
C08873=1072.808,-95.855,443.234,172.741,21.600,153.892
C08874=1072.801,-96.105,443.244,172.739,21.599,153.892
C08875=1072.796,-96.355,443.254,172.738,21.597,153.892
C08876=1072.790,-96.604,443.265,172.736,21.596,153.892
C08877=1072.784,-96.853,443.275,172.734,21.595,153.892
C08878=1072.777,-97.104,443.285,172.733,21.593,153.892
C08879=1072.772,-97.354,443.296,172.731,21.592,153.892
C08880=1072.765,-97.635,443.307,172.730,21.590,153.892
C08881=1072.758,-97.916,443.319,172.728,21.589,153.892
C08882=1072.751,-98.199,443.330,172.727,21.588,153.892
C08883=1072.744,-98.480,443.341,172.724,21.586,153.892
C08884=1072.738,-98.729,443.352,172.723,21.584,153.892
C08885=1072.732,-98.979,443.362,172.721,21.583,153.892
C08886=1072.725,-99.229,443.371,172.719,21.582,153.892
C08887=1072.720,-99.479,443.382,172.719,21.581,153.892
C08888=1072.714,-99.728,443.392,172.717,21.580,153.892
C08889=1072.707,-99.977,443.402,172.715,21.578,153.892
C08890=1072.702,-100.228,443.412,172.714,21.577,153.892
C08891=1072.695,-100.477,443.422,172.712,21.576,153.892
C08892=1072.688,-100.727,443.433,172.710,21.575,153.892
C08893=1072.683,-100.977,443.443,172.709,21.573,153.892
C08894=1072.676,-101.227,443.453,172.707,21.572,153.892
C08895=1072.670,-101.476,443.463,172.706,21.571,153.892
C08896=1072.665,-101.726,443.473,172.704,21.570,153.892
C08897=1072.658,-101.976,443.483,172.702,21.568,153.892
C08898=1072.652,-102.225,443.493,172.701,21.567,153.892
C08899=1072.647,-102.476,443.503,172.699,21.566,153.892
C08900=1072.640,-102.725,443.513,172.698,21.565,153.892
C08901=1072.634,-102.975,443.523,172.696,21.563,153.892
C08902=1072.628,-103.224,443.532,172.694,21.562,153.892
C08903=1072.622,-103.474,443.543,172.693,21.560,153.892
C08904=1072.616,-103.724,443.553,172.691,21.560,153.892
C08905=1072.610,-103.973,443.562,172.690,21.558,153.892
C08906=1072.603,-104.223,443.572,172.688,21.557,153.892
C08907=1072.598,-104.473,443.583,172.686,21.555,153.892
C08908=1072.592,-104.723,443.592,172.685,21.555,153.892
C08909=1072.585,-104.972,443.602,172.683,21.553,153.892
C08910=1072.579,-105.222,443.613,172.681,21.552,153.892
C08911=1072.573,-105.472,443.623,172.681,21.551,153.892
C08912=1072.567,-105.722,443.632,172.679,21.550,153.892
C08913=1072.560,-105.971,443.642,172.677,21.549,153.892
C08914=1072.554,-106.221,443.652,172.676,21.548,153.892
C08915=1072.549,-106.471,443.662,172.674,21.546,153.892
C08916=1072.543,-106.721,443.672,172.673,21.545,153.892
C08917=1072.536,-106.970,443.682,172.671,21.544,153.892
C08918=1072.530,-107.220,443.692,172.669,21.543,153.892
C08919=1072.525,-107.470,443.702,172.667,21.542,153.892
C08920=1072.518,-107.720,443.711,172.666,21.540,153.892
C08921=1072.512,-107.970,443.721,172.664,21.539,153.892
C08922=1072.506,-108.219,443.731,172.663,21.538,153.892
C08923=1072.500,-108.469,443.741,172.661,21.537,153.892
C08924=1072.493,-108.718,443.750,172.659,21.536,153.892
C08925=1072.487,-108.968,443.760,172.658,21.535,153.892
C08926=1072.481,-109.218,443.769,172.656,21.534,153.892
C08927=1072.475,-109.468,443.779,172.654,21.532,153.892
C08928=1072.469,-109.717,443.790,172.653,21.532,153.893
C08929=1072.463,-109.967,443.799,172.652,21.531,153.892
C08930=1072.457,-110.217,443.809,172.650,21.530,153.893
C08931=1072.451,-110.467,443.818,172.649,21.528,153.893
C08932=1072.445,-110.717,443.828,172.647,21.527,153.893
C08933=1072.438,-110.966,443.838,172.645,21.526,153.893
C08934=1072.432,-111.216,443.847,172.643,21.525,153.893
C08935=1072.426,-111.466,443.857,172.642,21.524,153.893
C08936=1072.420,-111.715,443.866,172.640,21.523,153.893
C08937=1072.414,-111.964,443.876,172.639,21.522,153.893
C08938=1072.408,-112.214,443.886,172.637,21.521,153.893
C08939=1072.402,-112.464,443.895,172.635,21.519,153.893
C08940=1072.396,-112.714,443.906,172.633,21.518,153.893
C08941=1072.390,-112.964,443.915,172.632,21.517,153.893
C08942=1072.384,-113.213,443.925,172.630,21.516,153.893
C08943=1072.378,-113.463,443.934,172.629,21.515,153.893
C08944=1072.370,-113.742,443.945,172.627,21.514,153.893
C08945=1072.364,-114.021,443.955,172.625,21.513,153.893
C08946=1072.357,-114.300,443.966,172.623,21.512,153.893
C08947=1072.349,-114.579,443.977,172.622,21.510,153.893
C08948=1072.343,-114.829,443.987,172.620,21.510,153.894
C08949=1072.337,-115.079,443.996,172.618,21.509,153.894
C08950=1072.332,-115.328,444.005,172.617,21.507,153.894
C08951=1072.325,-115.578,444.015,172.615,21.506,153.894
C08952=1072.319,-115.828,444.025,172.613,21.506,153.894
C08953=1072.313,-116.077,444.034,172.612,21.504,153.894
C08954=1072.307,-116.327,444.044,172.611,21.504,153.894
C08955=1072.301,-116.578,444.053,172.609,21.503,153.894
C08956=1072.295,-116.827,444.062,172.607,21.502,153.894
C08957=1072.289,-117.077,444.072,172.606,21.501,153.894
C08958=1072.282,-117.327,444.081,172.604,21.500,153.894
C08959=1072.276,-117.577,444.091,172.602,21.498,153.894
C08960=1072.270,-117.827,444.100,172.601,21.498,153.894
C08961=1072.265,-118.076,444.110,172.599,21.497,153.894
C08962=1072.258,-118.326,444.119,172.597,21.495,153.894
C08963=1072.252,-118.575,444.129,172.596,21.495,153.895
C08964=1072.246,-118.825,444.138,172.594,21.494,153.895
C08965=1072.239,-119.075,444.147,172.593,21.493,153.895
C08966=1072.233,-119.324,444.157,172.591,21.492,153.895
C08967=1072.227,-119.574,444.166,172.590,21.491,153.895
C08968=1072.221,-119.825,444.175,172.588,21.490,153.895
C08969=1072.215,-120.074,444.184,172.586,21.489,153.895
C08970=1072.209,-120.324,444.194,172.584,21.488,153.895
C08971=1072.203,-120.573,444.204,172.583,21.487,153.895
C08972=1072.197,-120.823,444.213,172.581,21.486,153.895
C08973=1072.191,-121.073,444.223,172.579,21.485,153.895
C08974=1072.184,-121.322,444.232,172.578,21.485,153.895
C08975=1072.178,-121.573,444.241,172.577,21.484,153.895
C08976=1072.172,-121.822,444.250,172.575,21.483,153.896
C08977=1072.166,-122.072,444.259,172.573,21.482,153.896
C08978=1072.160,-122.322,444.269,172.571,21.481,153.896
C08979=1072.154,-122.571,444.278,172.570,21.480,153.896
C08980=1072.148,-122.822,444.287,172.568,21.479,153.896
C08981=1072.141,-123.071,444.296,172.566,21.478,153.896
C08982=1072.135,-123.320,444.305,172.565,21.477,153.896
C08983=1072.129,-123.570,444.315,172.563,21.476,153.896
C08984=1072.123,-123.820,444.325,172.562,21.476,153.896
C08985=1072.117,-124.070,444.333,172.560,21.475,153.896
C08986=1072.110,-124.320,444.342,172.558,21.474,153.897
C08987=1072.105,-124.569,444.352,172.557,21.473,153.897
C08988=1072.099,-124.819,444.361,172.555,21.472,153.897
C08989=1072.093,-125.069,444.370,172.553,21.471,153.897
C08990=1072.086,-125.319,444.379,172.551,21.470,153.897
C08991=1072.080,-125.568,444.389,172.550,21.469,153.897
C08992=1072.073,-125.818,444.398,172.549,21.469,153.897
C08993=1072.068,-126.068,444.407,172.547,21.468,153.897
C08994=1072.061,-126.317,444.416,172.545,21.467,153.897
C08995=1072.055,-126.567,444.425,172.544,21.466,153.897
C08996=1072.049,-126.818,444.434,172.542,21.466,153.898
C08997=1072.043,-127.067,444.444,172.540,21.465,153.898
C08998=1072.037,-127.316,444.452,172.538,21.464,153.898
C08999=1072.031,-127.567,444.461,172.536,21.463,153.898
C09000=1072.024,-127.818,444.470,172.536,21.463,153.898
C09001=1072.019,-128.068,444.480,172.534,21.462,153.898
C09002=1072.016,-128.319,444.491,172.532,21.460,153.898
C09003=1072.014,-128.569,444.501,172.531,21.457,153.898
C09004=1072.015,-128.822,444.513,172.530,21.454,153.897
C09005=1072.019,-129.075,444.526,172.530,21.450,153.897
C09006=1072.024,-129.327,444.540,172.529,21.445,153.896
C09007=1072.032,-129.577,444.555,172.530,21.439,153.895
C09008=1071.641,-129.600,444.393,172.483,21.576,153.927
C09009=1071.632,-129.349,444.378,172.483,21.581,153.928
C09010=1071.627,-129.097,444.364,172.484,21.586,153.928
C09011=1071.624,-128.844,444.351,172.484,21.590,153.929
C09012=1071.623,-128.591,444.339,172.485,21.594,153.930
C09013=1071.624,-128.341,444.327,172.486,21.596,153.930
C09014=1071.627,-128.090,444.317,172.487,21.598,153.930
C09015=1071.632,-127.839,444.308,172.489,21.599,153.930
C09016=1071.638,-127.589,444.299,172.491,21.600,153.930
C09017=1071.645,-127.339,444.290,172.493,21.601,153.930
C09018=1071.651,-127.089,444.281,172.495,21.602,153.930
C09019=1071.657,-126.839,444.272,172.495,21.602,153.929
C09020=1071.663,-126.589,444.262,172.497,21.603,153.929
C09021=1071.669,-126.340,444.254,172.499,21.604,153.929
C09022=1071.675,-126.090,444.245,172.501,21.605,153.929
C09023=1071.681,-125.840,444.235,172.502,21.606,153.929
C09024=1071.688,-125.591,444.226,172.504,21.607,153.929
C09025=1071.694,-125.341,444.217,172.506,21.608,153.929
C09026=1071.700,-125.091,444.208,172.508,21.608,153.929
C09027=1071.706,-124.842,444.198,172.508,21.609,153.929
C09028=1071.713,-124.592,444.189,172.510,21.610,153.929
C09029=1071.718,-124.342,444.181,172.512,21.610,153.928
C09030=1071.725,-124.092,444.171,172.514,21.611,153.928
C09031=1071.731,-123.842,444.161,172.516,21.612,153.928
C09032=1071.736,-123.593,444.152,172.517,21.613,153.928
C09033=1071.743,-123.343,444.144,172.519,21.614,153.928
C09034=1071.749,-123.093,444.134,172.521,21.615,153.928
C09035=1071.755,-122.843,444.125,172.522,21.616,153.928
C09036=1071.762,-122.594,444.115,172.523,21.616,153.928
C09037=1071.768,-122.344,444.106,172.525,21.617,153.928
C09038=1071.773,-122.094,444.097,172.527,21.618,153.928
C09039=1071.780,-121.845,444.088,172.528,21.620,153.928
C09040=1071.786,-121.595,444.079,172.530,21.620,153.928
C09041=1071.792,-121.345,444.069,172.532,21.621,153.927
C09042=1071.798,-121.095,444.060,172.534,21.622,153.927
C09043=1071.805,-120.845,444.050,172.536,21.623,153.927
C09044=1071.810,-120.596,444.041,172.537,21.624,153.927
C09045=1071.816,-120.346,444.032,172.539,21.625,153.927
C09046=1071.822,-120.096,444.022,172.540,21.626,153.927
C09047=1071.829,-119.847,444.013,172.542,21.626,153.927
C09048=1071.835,-119.597,444.004,172.543,21.628,153.927
C09049=1071.841,-119.347,443.994,172.545,21.629,153.927
C09050=1071.848,-119.097,443.985,172.547,21.629,153.927
C09051=1071.854,-118.847,443.975,172.548,21.630,153.927
C09052=1071.859,-118.598,443.967,172.550,21.632,153.927
C09053=1071.865,-118.348,443.957,172.552,21.633,153.926
C09054=1071.871,-118.098,443.947,172.554,21.633,153.926
C09055=1071.878,-117.848,443.938,172.555,21.635,153.926
C09056=1071.884,-117.598,443.928,172.557,21.636,153.926
C09057=1071.890,-117.349,443.919,172.558,21.636,153.926
C09058=1071.897,-117.099,443.910,172.560,21.637,153.926
C09059=1071.903,-116.849,443.900,172.561,21.638,153.926
C09060=1071.909,-116.600,443.891,172.563,21.639,153.926
C09061=1071.915,-116.350,443.881,172.565,21.640,153.926
C09062=1071.921,-116.101,443.872,172.566,21.641,153.926
C09063=1071.927,-115.851,443.862,172.568,21.642,153.926
C09064=1071.933,-115.601,443.853,172.570,21.644,153.926
C09065=1071.939,-115.351,443.843,172.571,21.644,153.926
C09066=1071.946,-115.102,443.834,172.573,21.645,153.926
C09067=1071.952,-114.852,443.824,172.575,21.647,153.926
C09068=1071.958,-114.602,443.814,172.576,21.647,153.925
C09069=1071.964,-114.322,443.804,172.578,21.648,153.925
C09070=1071.971,-114.044,443.793,172.580,21.650,153.925
C09071=1071.978,-113.764,443.782,172.582,21.650,153.925
C09072=1071.985,-113.485,443.772,172.583,21.652,153.925
C09073=1071.991,-113.235,443.762,172.585,21.653,153.925
C09074=1071.997,-112.985,443.753,172.586,21.654,153.925
C09075=1072.004,-112.735,443.743,172.588,21.655,153.925
C09076=1072.010,-112.486,443.734,172.590,21.656,153.925
C09077=1072.016,-112.236,443.724,172.592,21.657,153.925
C09078=1072.022,-111.987,443.714,172.593,21.659,153.925
C09079=1072.028,-111.737,443.704,172.595,21.659,153.925
C09080=1072.034,-111.487,443.694,172.596,21.661,153.925
C09081=1072.040,-111.237,443.684,172.598,21.662,153.925
C09082=1072.046,-110.988,443.675,172.599,21.663,153.925
C09083=1072.052,-110.738,443.666,172.601,21.663,153.925
C09084=1072.058,-110.488,443.656,172.602,21.665,153.925
C09085=1072.064,-110.239,443.646,172.604,21.666,153.925
C09086=1072.070,-109.989,443.637,172.606,21.667,153.925
C09087=1072.077,-109.740,443.627,172.607,21.668,153.924
C09088=1072.083,-109.490,443.617,172.609,21.669,153.924
C09089=1072.089,-109.240,443.607,172.611,21.670,153.924
C09090=1072.095,-108.990,443.597,172.612,21.671,153.924
C09091=1072.101,-108.740,443.588,172.614,21.673,153.924
C09092=1072.107,-108.490,443.578,172.616,21.674,153.924
C09093=1072.114,-108.241,443.568,172.617,21.675,153.924
C09094=1072.120,-107.991,443.558,172.619,21.676,153.924
C09095=1072.126,-107.741,443.549,172.621,21.677,153.924
C09096=1072.132,-107.492,443.539,172.622,21.678,153.924
C09097=1072.138,-107.242,443.530,172.624,21.680,153.924
C09098=1072.144,-106.992,443.519,172.625,21.681,153.924
C09099=1072.150,-106.743,443.509,172.626,21.681,153.924
C09100=1072.156,-106.493,443.500,172.628,21.683,153.924
C09101=1072.162,-106.243,443.490,172.629,21.684,153.924
C09102=1072.169,-105.993,443.479,172.631,21.685,153.924
C09103=1072.175,-105.743,443.469,172.633,21.686,153.924
C09104=1072.181,-105.493,443.460,172.634,21.688,153.924
C09105=1072.187,-105.243,443.450,172.636,21.689,153.924
C09106=1072.193,-104.994,443.439,172.638,21.690,153.924
C09107=1072.199,-104.744,443.430,172.639,21.691,153.924
